PROPERTY FaultContactor : BOOL
GET
                    IF (Operational) THEN
	FaultContactor := lFaultContactor.Value;
ELSE
	FaultContactor := FALSE;	
END_IF
                  
END_GET
END_PROPERTY

PROPERTY FaultLevel : t_bms_fault_level
GET
                    IF (Operational) THEN
	FaultLevel := lFaultLevel.Value;
ELSE
	FaultLevel := cBMSFaultLevelNone;	
END_IF
                  
END_GET
END_PROPERTY

PROPERTY PackAverageTemperature : REAL
GET
                    PackAverageTemperature := lPackAverageTemperature.Value;

                  
END_GET
END_PROPERTY

PROPERTY PackChargeCurrent : REAL
GET
                    PackChargeCurrent := ABS(MIN(PackCurrent,0.0));


                  
END_GET
END_PROPERTY

PROPERTY PackChargeCurrentLimit : REAL
GET
                    IF (Operational) THEN // foobar should this be ValidTransmissions?
	PackChargeCurrentLimit := lPackChargeCurrentLimit.Value;
ELSE
	PackChargeCurrentLimit := 0.0;	
END_IF

                  
END_GET
END_PROPERTY

PROPERTY PackChargingCurrentTarget : REAL
GET
                    IF (Operational) THEN
	PackChargingCurrentTarget := lPackChargingCurrentTarget.Value;
ELSE
	PackChargingCurrentTarget := 0.0;	
END_IF


                  
END_GET
END_PROPERTY

PROPERTY PackChargingVoltageTarget : REAL
GET
                    PackChargingVoltageTarget := lPackChargingVoltageTarget.Value;

                  
END_GET
END_PROPERTY

PROPERTY PackCoolantTemperatureTarget : REAL
GET
                    PackCoolantTemperatureTarget := lPackCoolantTemperatureTarget.Value;
                  
END_GET
END_PROPERTY

PROPERTY PackCurrent : REAL
GET
                    IF (Operational) THEN
	PackCurrent := lPackCurrent.Value;
ELSE
	PackCurrent := 0.0;	
END_IF


                  
END_GET
END_PROPERTY

PROPERTY PackDischargeCurrent : REAL
GET
                    PackDischargeCurrent := MAX(PackCurrent,0.0);
                  
END_GET
END_PROPERTY

PROPERTY PackDischargeCurrentLimit : REAL
GET
                    IF (Operational) THEN
	PackDischargeCurrentLimit := lPackDischargeCurrentLimit.Value;
ELSE
	PackDischargeCurrentLimit := 0.0;	
END_IF


                  
END_GET
END_PROPERTY

PROPERTY PackFaultByte1 : USINT
GET
                    PackFaultByte1 := 0;
                  
END_GET
END_PROPERTY

PROPERTY PackFaultByte10 : USINT
GET
                    PackFaultByte10 := 0;
                  
END_GET
END_PROPERTY

PROPERTY PackFaultByte11 : USINT
GET
                    PackFaultByte11 := 0;
                  
END_GET
END_PROPERTY

PROPERTY PackFaultByte2 : USINT
GET
                    PackFaultByte2 := 0;
                  
END_GET
END_PROPERTY

PROPERTY PackFaultByte3 : USINT
GET
                    PackFaultByte3 := 0;
                  
END_GET
END_PROPERTY

PROPERTY PackFaultByte4 : USINT
GET
                    PackFaultByte4 := 0;
                  
END_GET
END_PROPERTY

PROPERTY PackFaultByte5 : USINT
GET
                    PackFaultByte5 := 0;
                  
END_GET
END_PROPERTY

PROPERTY PackFaultByte6 : USINT
GET
                    PackFaultByte6 := 0;
                  
END_GET
END_PROPERTY

PROPERTY PackFaultByte7 : USINT
GET
                    PackFaultByte7 := 0;
                  
END_GET
END_PROPERTY

PROPERTY PackFaultByte8 : USINT
GET
                    PackFaultByte8 := 0;
                  
END_GET
END_PROPERTY

PROPERTY PackFaultByte9 : USINT
GET
                    PackFaultByte9 := 0;
                  
END_GET
END_PROPERTY

PROPERTY PackFaultCode : USINT
GET
                    PackFaultCode := lPackFaultCode.Value;
                  
END_GET
END_PROPERTY

PROPERTY PackFaultNumber : USINT
GET
                    PackFaultNumber := lPackFaultNumber.Value;
                  
END_GET
END_PROPERTY

PROPERTY PackMaxTemperature : REAL
GET
                    PackMaxTemperature := lPackMaxTemperature.Value;
                  
END_GET
END_PROPERTY

PROPERTY PackMinTemperature : REAL
GET
                    PackMinTemperature := lPackMinTemperature.Value;
                  
END_GET
END_PROPERTY

PROPERTY PackSOC : t_percentage
GET
                    PackSOC := lPackSOC.Value;

                  
END_GET
END_PROPERTY

PROPERTY PackSOH : t_percentage
GET
                    PackSOH := lPackSOH.Value;
                  
END_GET
END_PROPERTY

PROPERTY PackTotalChargeEnergy : REAL
GET
                    PackTotalChargeEnergy := lPackTotalChargeEnergy.Value;
                  
END_GET
END_PROPERTY

PROPERTY PackTotalDischargeEnergy : REAL
GET
                    PackTotalDischargeEnergy := lPackTotalDischargeEnergy.Value;
                  
END_GET
END_PROPERTY

PROPERTY PackVoltage : REAL
GET
                    PackVoltage := lPackVoltage.Value;
                  
END_GET
END_PROPERTY

PROPERTY RequestDisconnect : BOOL
GET
                    RequestDisconnect := lRequestDisconnect.Value;
                  
END_GET
END_PROPERTY

PROPERTY RequestedBMSChargeState : t_bms_charge_state
GET
                    RequestedBMSChargeState := lRequestedBMSChargeState.Value;

                  
END_GET
SET
                    lRequestedBMSChargeState.Value := RequestedBMSChargeState;

                  
END_SET
END_PROPERTY

PROPERTY RequestedBMSState : t_bms_state
GET
                    RequestedBMSState := lRequestedBMSState.Value;
                  
END_GET
SET
                    lRequestedBMSState.Value := RequestedBMSState;


                  
END_SET
END_PROPERTY

PROPERTY RequestedTMSState : t_tms_state
GET
                    IF (Operational) THEN
	RequestedTMSState := lRequestedTMSState.Value;
ELSE
	RequestedTMSState := cTMSStateShutdown;	
END_IF
                  
END_GET
END_PROPERTY

PROPERTY TypeToken : t_medium_string
GET
                    TypeToken := 'cBMS';
                  
END_GET
END_PROPERTY

PROPERTY Peripheral : REFERENCE TO Peripheral
GET
                    Peripheral ref= lPeripheral;
                  
END_GET
END_PROPERTY
END_FUNCTION_BLOCK

FUNCTION_BLOCK ControllerCharger EXTENDS MimicCANOpenSlave
  VAR CONSTANT
    cChargingCurrentPhysicalMaxACSinglePhase : REAL := 38.0;  (* foobar changed from 48, CATL needs to allow higher values *)
    cOBCStatusPeriod : t_time := TIME#2s0ms;
  END_VAR
  VAR
    lChargingVoltageMax : ValueObjectRealOffsetScaledOutputReferenceUINTSwitched;
    lChargingCurrentMax : ValueObjectRealOffsetScaledOutputReferenceUINTSwitched;
    lHeatingMode : ValueObjectBoolOutputReferenceUSINT;
    lStopCharging : ValueObjectBoolOutputReferenceUSINT;
    lVoltage : ValueObjectRealScaledOffsetInputReferenceUINTSwitched;
    lCurrent : ValueObjectRealScaledOffsetInputReferenceUINTSwitched;
    lPower : ValueObjectRealScaledOffsetInputReferenceUSINT;
    lDiagnosticState : ValueObjectUINTInputReferenceUINT;
    lOBCStatus : ValueObjectEnumTypeInputReferenceUINT;
    lStatusCC : ValueObjectBoolInputReferenceUINT;
    lStatusCP : ValueObjectBoolInputReferenceUINT;
    lCurrentOBCState : ValueObjectEnumType;
    lRequestedOBCState : ValueObjectEnumType;
    lIgnoreOBCStatusNone : BOOL := TRUE;
    lChargingCurrentPhysicalMax : REAL := cChargingCurrentPhysicalMaxACSinglePhase;  (* foobar *)
    lOBCStatusTimer : t_timer;
    lOBCStatusDerived : t_obc_status;
  END_VAR

            ;
          

METHOD initialize
                  lChargingVoltageMax.Offset := 0.0;
lChargingVoltageMax.Scaling := 10.0;
lChargingVoltageMax.initializeValueObjectOp(OpSelf,'TargVoltage','Onboard charger target voltage','volts',cValueStyleConfigurable);

lChargingCurrentMax.Offset := 0.0;
lChargingCurrentMax.Scaling := 10.0;
lChargingCurrentMax.initializeValueObjectOp(OpSelf,'TargCurrent','Onboard charger target current','amps',cValueStyleConfigurable);

lHeatingMode.Index := 0;
lHeatingMode.initializeValueObjectOp(OpSelf,'Heating','Onboard charger heating mode','',cValueStyleConfigurable);

lStopCharging.Index := 0;
lStopCharging.initializeValueObjectOp(OpSelf,'Stop','Onboard charger stop status','',cValueStyleConfigurable);

lVoltage.Offset := 0.0;
lVoltage.Scaling := 0.1;
lVoltage.initializeValueObjectOp(OpSelf,'Voltage','Onboard charger measured voltage','volts',cValueStyleConfigurable);

lCurrent.Offset := 0.0;
lCurrent.Scaling := 0.1;
lCurrent.initializeValueObjectOp(OpSelf,'Current','Onboard charger measured current','amps',cValueStyleConfigurable);

lPower.Offset := 0.0;
lPower.Scaling := 100.0;
lPower.initializeValueObjectOp(OpSelf,'Power','Onboard charger measured power','kW',cValueStyleConfigurable);

lDiagnosticState.initializeValueObjectOp(OpSelf,'Diagnostic','Onboard charger current diagnostic','',cValueStyleConfigurable);

lStatusCC.Index := 5;
lStatusCC.initializeValueObjectOp(OpSelf,'CC','Onboard charger CC signal','',cValueStyleConfigurable);
lStatusCC.InputReference REF= lDiagnosticState.ValueReference;

lStatusCP.Index := 6;
lStatusCP.initializeValueObjectOp(OpSelf,'CP','Onboard charger CP signal','',cValueStyleConfigurable);
lStatusCP.InputReference REF= lDiagnosticState.ValueReference;

lOBCStatus.Index := 8;
lOBCStatus.Length := 2;
lOBCStatus.EnumType := cEnumTypeOBCStatus;
lOBCStatus.initializeValueObjectOp(OpSelf,'OBCStatus','Onboard charger OBC status','',cValueStyleConfigurable);
lOBCStatus.InputReference REF= lDiagnosticState.ValueReference;

lCurrentOBCState.EnumType := cEnumTypeOBCState;
lCurrentOBCState.initializeValueObject(NopSelf,'CrrOBCStt','Onboard charger current OBC state','',cValueStyleConfigurable);

lRequestedOBCState.EnumType := cEnumTypeOBCState;
lRequestedOBCState.initializeValueObject(NopSelf,'ReqOBCStt','Onboard charger requested OBC state','',cValueStyleConfigurable);
	
SUPER^.initialize();
SubSystem := cSubsystemBattery;

lAlarmCANOpenSlaveNotOperational.InitialSeverity := cSeverityNone;
lAlarmCANOpenSlaveNotOperational.SeverityWarningTimeout := T#250MS;
lAlarmCANOpenSlaveNotOperational.SeverityErrorTimeout := T#1S;
lAlarmCANOpenSlaveNotOperational.SeverityCriticalTimeout := T#5S;

lAlarmCANOpenSlaveAllowableUp.AllowableSystemState := cSystemStatePreparing;
lAlarmCANOpenSlaveAllowableUp.UpperSystemStateScope := cSystemStatePreparing;
lAlarmCANOpenSlaveAllowableUp.LowerSystemStateScope := cSystemStatePreparing;

lStartSystemStateScope := t_system_state.cSystemStatePreparing;
lOperationalSystemStateScopeLower := t_system_state.cSystemStateCharging;
lModulationSystemStateScope := t_system_state.cSystemStateCharging;

lModulationSeverity := cSeverityError; // foobar default or not?

lOBCStatusTimer.initialize();
lOBCStatusTimer.Enable := TRUE;
lOBCStatusTimer.Period := cOBCStatusPeriod;


                
END_METHOD

METHOD operator
                  SUPER^.operator();

setCurrentOBCState();

HeatingMode := FALSE;

CASE (RequestedOBCState) OF
	cOBCStateDisconnected:
		StopCharging := TRUE;	
	cOBCStateCharging:
		StopCharging := FALSE;
	cOBCStateStandby:
		StopCharging := TRUE;
	cOBCStateError:
		StopCharging := TRUE;
END_CASE

// lFaultHardware.Index := 0; 16#1
// lFaultTemperature.Index := 1; 16#2
// lFaultInputVoltage.Index := 2; 16#4
// lFaultBattery.Index := 3; 16#8
// lFaultCommunications.Index := 4; 16#10
// lWarningTemperature.Index := 14; 16#4000

// lStatusSwitch.Index := 12;
// lStatusFan.Index := 15;

IF (WORD_TO_BOOL(UINT_TO_WORD(lDiagnosticState.Value) AND 16#401F)) THEN
	lAlarmCANOpenSlaveNotify.triggerWithContext(UINT_TO_WORD(lDiagnosticState.Value));
END_IF


                
END_METHOD

METHOD setCurrentOBCState
                  IF (NOT(Operational)) THEN
	CurrentOBCState := cOBCStateDisconnected;
	RETURN;
END_IF

IF (OBCStatus<>cOBCStatusNone) THEN
	lOBCStatusTimer.reset();
END_IF
lOBCStatusTimer.operator();

IF (((NOT(lOBCStatusTimer.Expired)) OR
	(lIgnoreOBCStatusNone)) AND
	(OBCStatus=cOBCStatusNone)) THEN
	lOBCStatusDerived := cOBCStatusStandby ;
ELSE
	lOBCStatusDerived := OBCStatus;
END_IF

IF (lOBCStatusDerived=cOBCStatusNone) THEN
	CurrentOBCState := cOBCStateDisconnected;
	RETURN;
END_IF

IF (StatusCC) THEN
	CurrentOBCState := cOBCStateDisconnected;
	RETURN;
END_IF

CurrentOBCState := cOBCStateStandby;

IF ((NOT(StatusCC)) AND (StatusCP)) THEN
	// foobar not powered on
	RETURN;
END_IF

IF ((NOT(StatusCP)) AND
	(NOT(StatusCC)) AND
	(OBCStatus=cOBCStatusCharging) AND
	(lEnabled)) THEN
	CurrentOBCState := cOBCStateCharging;
END_IF

IF (OBCStatus=cOBCStatusError) THEN
	CurrentOBCState := cOBCStateError;
END_IF

                
END_METHOD

METHOD initializeCharger
  VAR_INPUT
    voltage : REFERENCE TO UINT;
    current : REFERENCE TO UINT;
    power : REFERENCE TO USINT;
    status : REFERENCE TO UINT;
    chargingVoltageMax : REFERENCE TO UINT;
    chargingCurrentMax : REFERENCE TO UINT;
    mode : REFERENCE TO USINT;
    command : REFERENCE TO USINT;
  END_VAR
                  lVoltage.InputReference REF= voltage;
lCurrent.InputReference REF= current;
lPower.InputReference REF= power;
lDiagnosticState.InputReference REF= status;

lChargingVoltageMax.OutputReference REF= chargingVoltageMax;
lChargingCurrentMax.OutputReference REF= chargingCurrentMax;
lHeatingMode.OutputReference REF= mode;
lStopCharging.OutputReference REF= command;

                
END_METHOD

PROPERTY ChargingCurrentMax : REAL
GET
                    ChargingCurrentMax := lChargingCurrentMax.Value;

                  
END_GET
SET
                    lChargingCurrentMax.Value := MIN(ChargingCurrentMax,lChargingCurrentPhysicalMax);
                  
END_SET
END_PROPERTY

PROPERTY ChargingVoltageMax : REAL
GET
                    ChargingVoltageMax := lChargingVoltageMax.Value;

                  
END_GET
SET
                    lChargingVoltageMax.Value := ChargingVoltageMax;
                  
END_SET
END_PROPERTY

PROPERTY Current : REAL
GET
                    Current := lCurrent.Value;

                  
END_GET
END_PROPERTY

PROPERTY CurrentOBCState : t_obc_state
GET
                    lCurrentOBCState.operator();
CurrentOBCState := lCurrentOBCState.Value;

                  
END_GET
SET
                    lCurrentOBCState.Value := CurrentOBCState;
                  
END_SET
END_PROPERTY

PROPERTY HeatingMode : BOOL
GET
                    HeatingMode := lHeatingMode.Value;

                  
END_GET
SET
                    lHeatingMode.Value := HeatingMode;
                  
END_SET
END_PROPERTY

(* {attribute 'monitoring' := 'call'} *)
PROPERTY OBCStatus : t_obc_status
GET
                    OBCStatus := lOBCStatus.Value;

                  
END_GET
END_PROPERTY

PROPERTY Power : REAL
GET
                    Power := lPower.Value;

                  
END_GET
END_PROPERTY

PROPERTY RequestedOBCState : t_obc_state
GET
                    lRequestedOBCState.operator();
RequestedOBCState := lRequestedOBCState.Value;
                  
END_GET
SET
                    lRequestedOBCState.Value := RequestedOBCState;


                  
END_SET
END_PROPERTY

(* {attribute 'monitoring' := 'call'} *)
PROPERTY StatusCC : BOOL
GET
                    StatusCC := lStatusCC.Value;

                  
END_GET
END_PROPERTY

(* {attribute 'monitoring' := 'call'} *)
PROPERTY StatusCP : BOOL
GET
                    StatusCP := lStatusCP.Value;

                  
END_GET
END_PROPERTY

PROPERTY StopCharging : BOOL
GET
                    StopCharging := lStopCharging.Value;

                  
END_GET
SET
                    lStopCharging.Value := StopCharging;

                  
END_SET
END_PROPERTY

PROPERTY TypeToken : t_medium_string
GET
                    TypeToken := 'cCharger';
                  
END_GET
END_PROPERTY

PROPERTY Voltage : REAL
GET
                    Voltage := lVoltage.Value;

                  
END_GET
END_PROPERTY
END_FUNCTION_BLOCK

FUNCTION_BLOCK ControllerChargerSlave EXTENDS ControllerCharger

            ;
          

METHOD initialize
                  SUPER^.initialize();

// invalid scope as only ChargerA controls AllowUp
lAlarmCANOpenSlaveAllowableUp.AllowableSystemState := cSystemStateCharging;
lAlarmCANOpenSlaveAllowableUp.UpperSystemStateScope := cSystemStateStandby;
lAlarmCANOpenSlaveAllowableUp.LowerSystemStateScope := cSystemStatePreparing;

lOperationalSystemStateScopeLower := t_system_state.cSystemStateCharging;
lOperationalSystemStateScopeUpper := t_system_state.cSystemStateCharging;

                
END_METHOD
END_FUNCTION_BLOCK

{attribute 'enable_dynamic_creation'}
FUNCTION_BLOCK ControllerMotor EXTENDS CANOpenSlave
  VAR_INPUT
    lRequestedThrottle : ValueObjectPercentage;
    lTypeSteer : BOOL := FALSE;
    lMaximumVelocity : REAL := 50.0;
    lAutomaticEnable : BOOL := TRUE;
    lAlwaysEnable : BOOL := FALSE;
  END_VAR
  VAR CONSTANT
    cStallPeriod : t_time := TIME#1s0ms;
    cNominalVoltage : REAL := 120.0;
    cTorquePeriod : t_time := TIME#250ms;
    cThrottleArbitrationAllowableDelta : t_percentage := 0.15;
    cThrottleArbitrationThreshold : t_percentage := 0.25;
    cThrottleArbitrationPeriod : t_time := TIME#2s0ms;
    cThrottleThreshold : t_percentage := 0.001;
    cThrottleFreeWheelThreshold : t_percentage := 0.002;
    cNMTDetectionPeriod : t_time := TIME#250ms;
    cEnabledPeriod : t_time := TIME#20s0ms;
    cMotorTemperatureType : DWORD := 4;
    cInitializeMotorHoldCount : USINT := 2;
    cInitializeMotorHoldPeriod : t_time := TIME#7s0ms;
    cNominalCurrent400A : REAL := 400.0;
    cPolePairs400A : REAL := 3.0;
    cControllerTemperatureInitialCutbackThreshold400A : REAL := 75.0;
    cControllerTemperatureCutoutThreshold400A : REAL := 100.0;
    cControllerTemperatureMinimumThreshold400A : t_percentage := 0.2;
    cMotorTemperatureInitialCutbackThreshold400A : REAL := 110.0;
    cMotorTemperatureCutoutThreshold400A : REAL := 160.0;
    cMotorTemperatureMinimumThreshold400A : t_percentage := 0.2;
    cMotorTemperatureInvalidRange400A : REAL := 200;
    cNominalCurrent150A : REAL := 150.0;
    cPolePairs150A : REAL := 2.0;
    cControllerTemperatureInitialCutbackThreshold150A : REAL := 75.0;
    cControllerTemperatureCutoutThreshold150A : REAL := 80.0;
    cControllerTemperatureMinimumThreshold150A : t_percentage := 0.2;
    cMotorTemperatureInitialCutbackThreshold150A : REAL := 110.0;
    cMotorTemperatureCutoutThreshold150A : REAL := 120.0;
    cMotorTemperatureMinimumThreshold150A : t_percentage := 0.2;
    cMotorTemperatureInvalidRange150A : REAL := 200;
  END_VAR
  VAR
    lVREnableStallAutomaticClearing : ValueReferenceBool;
    lEnableStallAutomaticClearing : BOOL := TRUE;
    lVREnableStallResponse : ValueReferenceBool;
    lEnableStallResponse : BOOL := FALSE;
    lVREnableHoldStationary : ValueReferenceBool;
    lEnableHoldStationary : BOOL := FALSE;
    lVREnableStallDetection : ValueReferenceBool;
    lEnableStallDetection : BOOL := FALSE;
    lVREnableThrottleArbitration : ValueReferenceBool;
    lEnableThrottleArbitration : BOOL := FALSE;
    lVREnableNMTDetectionTPDO : ValueReferenceBool;
    lEnableNMTDetectionTPDO : BOOL := FALSE;
    lVREnableInitializeHold : ValueReferenceBool;
    lEnableInitializeHold : BOOL := FALSE;
    lAlarmControllerTemperatureCutback : CutbackInterlock;
    lAlarmMotorTemperatureCutback : CutbackInterlock;
    lAlarmMotorTemperatureSensor : ReportableAlarm;
    lTargetSpeed : ValueObjectRealScaledOffsetOutputUINT;
    lEnable : ValueObjectBoolOutputUINT;
    lForward : ValueObjectBoolOutputUINT;
    lReverse : ValueObjectBoolOutputUINT;
    lClearAlarm : ValueObjectBoolOutputUINT;
    lVelocity : ValueObjectRealScaledOffsetInputReferenceINT;
    lTPDO1Stuffing : ValueObjectBoolInputReferenceUINT;
    lCurrent : ValueObjectRealScaledOffsetInputReferenceUSINT;
    lAlarm : ValueObjectUINTInputReferenceUINT;  (* foobar *)
    lMotorTemperature : ValueObjectRealScaledOffsetInputReferenceUSINT;
    lControllerTemperature : ValueObjectRealScaledOffsetInputReferenceSINT;
    lBatteryCurrent : ValueObjectRealScaledOffsetInputReferenceUSINT;
    lBatteryVoltage : ValueObjectRealScaledOffsetInputReferenceUINT;
    lBatteryPower : ValueObjectRealScaledOffset;
    lTorque : ValueObjectRealScaledOffsetInputUINT;  (* foobar *)
    lMotorTemperatureEnableCANSequence : MotorTemperatureEnableCANSequence;
    lCheckMotorTemperatureEnableCANMessage : CheckMotorTemperatureEnableCANMessage;
    lEnableRPDO1 : BOOL := TRUE;
    lTargetVelocity : REAL;
    lControl : WORD;
    lTorqueTimer : t_timer;
    lMotorTemperatureInvalidRange : REAL;
    lMotorTemperatureSensorRecovery : REAL;
    lEnableDiscriminatoryMotorTemperatureControl : BOOL := FALSE;  (* foobar *)
    lMotorTemperatureEnabled : BOOL := TRUE;
    lMotorTemperatureEnabledVerified : BOOL := FALSE;
    lHoldStationary : BOOL := FALSE;  (* lMaximumVelocity: REAL:= 50.0; lAutomaticEnable: BOOL:= TRUE; lAlwaysEnable: BOOL:= FALSE; *)
    lEnabledTimer : t_timer;
    lInitializeMotorHoldCounter : USINT := 0;
    lInitializeMotorHoldTimer : t_timer;
    lEnableFreeWheel : BOOL := FALSE;
    lFreeWheel : BOOL := FALSE;
    lDiagnostic : t_motor_diagnostic;
    _Diagnostic : t_motor_diagnostic;
    lStallTimer : t_timer;
    lStallState : t_stall_state := cStallStateNone;
    lStalled : BOOL := FALSE;
    lStallInput : BOOL := FALSE;
    lStalledCount : USINT := 0;
    lStationary : BOOL := FALSE;
    lTargetSpeedIndicator : USINT := 0;
    lZeroTargetSpeedIndicator : USINT := 0;
    lCurrentVelocityIndicator : USINT := 0;
    lZeroCurrentVelocityIndicator : USINT := 0;
    lStallIndicator : USINT := 0;
    lNoStallIndicator : USINT := 0;
    lStalledIndicator : USINT := 0;
    lNotStalledIndicator : USINT := 0;
    lRPDO1Message : T_x_can_msg;
    lSyncAlternateState : BOOL;
    lSDOTorque : CIA405.SDO_READ_DATA;
    lSDOTorqueData : DWORD;
    lSDOTorqueLastSuccessfulReadData : DWORD;
    lSDOTorqueDataLength : UDINT := 4;
    lSDOTorqueSuccess : BOOL := FALSE;
    lSDOTorqueAttemptCounter : USINT := 0;
    lSDOTorqueSuccessCounter : USINT := 0;
    lNominalVoltage : REAL := cNominalVoltage;
    lNominalCurrent : REAL := 0.0;
    lPolePairs : REAL := 1.0;
    lThrottleThreshold : t_percentage := cThrottleThreshold;
    lThrottleFreeWheelThreshold : t_percentage := cThrottleFreeWheelThreshold;
    lRequestedThrottlePrevious : t_percentage;
    lProposedThrottle : t_percentage;
    lMeasuredThrottle : t_percentage;
    lThrottleArbitrationDelta : t_percentage;
    lThrottleArbitrationAllowableDelta : t_percentage := cThrottleArbitrationAllowableDelta;
    lThrottleArbitrationThreshold : t_percentage := cThrottleArbitrationThreshold;
    lThrottleArbitrationTimer : t_timer;
    lRPDO1Alternate : BOOL := TRUE;
    lNMTDetectionTimer : t_timer;
    lTPDO1StuffingPrevious : BOOL;
  END_VAR

            ;
          

METHOD cancelSDOTorque
                  lSDOTorque.ENABLE := FALSE;
lSDOTorqueDataLength := 4;
lSDOTorque(DATALENGTH:=lSDOTorqueDataLength);

                
END_METHOD

METHOD checkMotorTemperatureEnabled
                  //requestSDORead(TRUE,16#20F1,2,4);

IF (lCheckMotorTemperatureEnableCANMessage.Success) THEN
	lMotorTemperatureEnabledVerified := TRUE;
	lMotorTemperatureEnabled := lCheckMotorTemperatureEnableCANMessage.MotorTemperatureEnabled;
	lCheckMotorTemperatureEnableCANMessage.reset();
	RETURN;
END_IF

IF (NOT(lCheckMotorTemperatureEnableCANMessage.Running)) THEN
	lCheckMotorTemperatureEnableCANMessage.start();
END_IF


                
END_METHOD

METHOD emergencyHandler
  VAR_INPUT
    info : t_canopen_emcy;
  END_VAR
  VAR
    eid : t_motor_emcy_id;
    first : BOOL;
  END_VAR
                  first := emergencyRegisterAdd(info);

eid := WORD_TO_INT(info.EMCY_ERROR_CODE);

CASE eid OF
	t_motor_emcy_id.cEMCY_none:
		RETURN;

	t_motor_emcy_id.cEMCY_CONTACTOR_OPEN,
	t_motor_emcy_id.cEMCY_CONTACTOR_CLOSED,
	t_motor_emcy_id.cEMCY_PUMP_VMN_LOW,
	t_motor_emcy_id.cEMCY_PUMP_VMN_HIGH,
	t_motor_emcy_id.cEMCY_TILLER_ERROR,
	t_motor_emcy_id.cEMCY_PUMP_VMN_NOT_OK,
	t_motor_emcy_id.cEMCY_HVIL_FAIL,
	t_motor_emcy_id.cEMCY_SEAT_MISMATCH,
	t_motor_emcy_id.cEMCY_PEDAL_WIRE_KO,
	t_motor_emcy_id.cEMCY_PUMP_VACC_NOT_OK,
	t_motor_emcy_id.cEMCY_PUMP_INC_START,
	t_motor_emcy_id.cEMCY_PUMP_VACC_RANGE,
	t_motor_emcy_id.cEMCY_HANDBRAKE:
		lAlarmCANOpenSlaveNotify.triggerWithContext(INT_TO_LWORD(eid));
		RETURN;
				
	t_motor_emcy_id.cEMCY_MC_EB_COIL_SHORT,
	t_motor_emcy_id.cEMCY_DRIVER_SHORTED,
	t_motor_emcy_id.cEMCY_CONTACTOR_DRIVER,
	t_motor_emcy_id.cEMCY_EVP_DRIV_SHORT,
	t_motor_emcy_id.cEMCY_EVP_COIL_SHORT,
	t_motor_emcy_id.cEMCY_EVP2_COIL_SHORT,
	t_motor_emcy_id.cEMCY_HW_FAULT_MC,
	t_motor_emcy_id.cEMCY_POSITIVE_LC_OPEN,
	t_motor_emcy_id.cEMCY_LC_COIL_OPEN,
	t_motor_emcy_id.cEMCY_CONTROLLER_MISM,
	t_motor_emcy_id.cEMCY_NO_CAN_MSG,
	t_motor_emcy_id.cEMCY_WRONG_SET_BAT,
	t_motor_emcy_id.cEMCY_WRONG_KEY_VOLT,
	t_motor_emcy_id.cEMCY_CAPACITOR_CHARGE,
	t_motor_emcy_id.cEMCY_WRONG_FBSENSSET,
	t_motor_emcy_id.cEMCY_OFFSET_SPDSENS,
	t_motor_emcy_id.cEMCY_SPEED_OVERHEAD,
	t_motor_emcy_id.cEMCY_WRONG_RAM_MEM,
	t_motor_emcy_id.cEMCY_POWER_MISMATCH,
	t_motor_emcy_id.cEMCY_IQ_MISMATCHED,
	t_motor_emcy_id.cEMCY_FIELD_ORIENT_KO,
	t_motor_emcy_id.cEMCY_WATCHDOG,
	t_motor_emcy_id.cEMCY_SAFETY_INIT_XX,
	t_motor_emcy_id.cEMCY_SAFETY_SW_XX,
	t_motor_emcy_id.cEMCY_SAFETY_DIAG_XX,
	t_motor_emcy_id.cEMCY_STBY_HIGH,
	t_motor_emcy_id.cEMCY_VMN_HIGH,
	t_motor_emcy_id.cEMCY_INIT_VMN_HIGH,
	t_motor_emcy_id.cEMCY_VMN_LOW,
	t_motor_emcy_id.cEMCY_INIT_VMN_LOW,
	t_motor_emcy_id.cEMCY_POS_EB_SHORTED,
	t_motor_emcy_id.cEMCY_SMARTDRIVER_KO,
	t_motor_emcy_id.cEMCY_AUX_BATT_SHORT,
	t_motor_emcy_id.cEMCY_VKEY_OFF_SHORTED,
	t_motor_emcy_id.cEMCY_LOGIC_FAILURE_1,
	t_motor_emcy_id.cEMCY_LOGIC_FAILURE_3,
	t_motor_emcy_id.cEMCY_LOGIC_FAILURE_2,
	t_motor_emcy_id.cEMCY_SENSOR_SUPPLY_XX,
	t_motor_emcy_id.cEMCY_POSEBSHORT_PIN,
	t_motor_emcy_id.cEMCY_ED_SLIP_MISMATCH,
	t_motor_emcy_id.cEMCY_POSEBSHORT_GND,
	t_motor_emcy_id.cEMCY_SHORT_CIRCUIT_KO,
	t_motor_emcy_id.cEMCY_SHORT_CIRCUIT,
	t_motor_emcy_id.cEMCY_IMS_ERROR,
	t_motor_emcy_id.cEMCY_SPEED_FBERR_XX,
	t_motor_emcy_id.cEMCY_MOTPHASE_SH,
	t_motor_emcy_id.cEMCY_VDC_OFF_SHORTED,
	t_motor_emcy_id.cEMCY_HW_FAULT,
	t_motor_emcy_id.cEMCY_POWERMOS_SHORTED,
	t_motor_emcy_id.cEMCY_CTRAP_THRESHOLD,
	t_motor_emcy_id.cEMCY_OUT_MISMATCH_PU,
	t_motor_emcy_id.cEMCY_SP_MISMATCH_XX,
	t_motor_emcy_id.cEMCY_ANALOG_INPUT,
	t_motor_emcy_id.cEMCY_OVERLOAD,
	t_motor_emcy_id.cEMCY_VDC_LINK_OVERV:
		lAlarmCANOpenSlaveBlock.triggerWithContext(INT_TO_LWORD(eid));
		RETURN;
		
	t_motor_emcy_id.cEMCY_EB_DRIVSHRT,
	t_motor_emcy_id.cEMCY_EB_DRIVOPEN,
	t_motor_emcy_id.cEMCY_EVP_COIL_OPEN,
	t_motor_emcy_id.cEMCY_VACC_NOT_OK,
	t_motor_emcy_id.cEMCY_BMS_NOT_READY,
	t_motor_emcy_id.cEMCY_POT_MISMATCH,
	t_motor_emcy_id.cEMCY_AGV,
	t_motor_emcy_id.cEMCY_REMA_T_ALARM,
	t_motor_emcy_id.cEMCY_SENS_BAT_TEMP_KO,
	t_motor_emcy_id.cEMCY_EMERGENCY,
	t_motor_emcy_id.cEMCY_LIFT_LOWER,
	t_motor_emcy_id.cEMCY_PARAM_TRANSFER,
	t_motor_emcy_id.cEMCY_EPS_RELAY_OPEN,
	t_motor_emcy_id.cEMCY_EB_COIL_OPEN,
	t_motor_emcy_id.cEMCY_PEB_PEVP_NOT_OK,
	t_motor_emcy_id.cEMCY_PEV_NOT_OK,
	t_motor_emcy_id.cEMCY_VACC_OUT_RANGE,
	t_motor_emcy_id.cEMCY_HW_FAULT_EB,
	t_motor_emcy_id.cEMCY_CONT_DRV_EV,
	t_motor_emcy_id.cEMCY_COIL_SHOR_EVAUX,
	t_motor_emcy_id.cEMCY_EVP_DRIVER_OPEN,
	t_motor_emcy_id.cEMCY_DRV_SHOR_EV,
	t_motor_emcy_id.cEMCY_NO_CAN_WR_MSGXX,
	t_motor_emcy_id.cEMCY_STO_SS1_ALARM_XX,
	t_motor_emcy_id.cEMCY_WRONG_PERFORM,
	t_motor_emcy_id.cEMCY_WRONG_SLAVE_VER,
	t_motor_emcy_id.cEMCY_MS_PAR_CHK_MISM,
	t_motor_emcy_id.cEMCY_CURRENT_PROFILE,
	t_motor_emcy_id.cEMCY_EEPROM_KO,
	t_motor_emcy_id.cEMCY_COIL_SHOR_EB,
	t_motor_emcy_id.cEMCY_STO_SS1_ACTIVEXX,
	t_motor_emcy_id.cEMCY_RPM_HIGH,
	t_motor_emcy_id.cEMCY_STALL_ROTOR,
	t_motor_emcy_id.cEMCY_INCORRECT_START,
	t_motor_emcy_id.cEMCY_FORW_BACK,
	t_motor_emcy_id.cEMCY_MOTOR_TEMP_STOP:
		lAlarmCANOpenSlaveBlock.triggerWithContext(INT_TO_LWORD(eid));
		IF (first) THEN
			lAlarmCANOpenSlaveStop.triggerWithContext(INT_TO_LWORD(eid));
		END_IF
	
		RETURN;
		
	t_motor_emcy_id.cEMCY_THERMIC_SENS_KO,
	t_motor_emcy_id.cEMCY_THERMPUSENSKO,
	t_motor_emcy_id.cEMCY_SENS_MOT_TEMP_KO:
		lAlarmCANOpenSlaveBlock.triggerWithContext(INT_TO_LWORD(eid));; //foobar disable remedy
		RETURN;
END_CASE

lAlarmCANOpenSlaveNotify.triggerWithContext(INT_TO_LWORD(eid));

	//t_motor_emcy_id.cEMCY_REMA_T_ALARM,								//duplicate id
	//	lAlarmCANOpenStop.triggerWithContext(eid);

	//t_motor_emcy_id.cEMCY_SP_MISMATCH_PUMP,                     //duplicate id
	//	lAlarmCANOpenSlaveBlock.triggerWithContext(eid);
	
	//t_motor_emcy_id.cEMCY_OPEN_COIL_EV,							//duplicate id
	//	lAlarmCANOpenStop.triggerWithContext(eid);
	
	//t_motor_emcy_id.cEMCY_WRONG_FBSENSSET,					//duplicate id
	//	lAlarmCANOpenSlaveBlock.triggerWithContext(eid);
		
	//t_motor_emcy_id.cEMCY_WSET_TG_EB_XX,						//duplicate id
	//	lAlarmCANOpenSlaveBlock.triggerWithContext(eid);
	
	//t_motor_emcy_id.cEMCY_INPUT_MISMATCH,						//duplicate id
	//	lAlarmCANOpenSlaveBlock.triggerWithContext(eid);
		
	//t_motor_emcy_id.cEMCY_SAFETY_DIAG_XX,						//duplicate
	//	lAlarmCANOpenSlaveBlock.triggerWithContext(eid);
	
	//t_motor_emcy_id.cEMCY_SAFETY_SW_XX,							//duplicate
	//	lAlarmCANOpenSlaveBlock.triggerWithContext(eid);
	
	//t_motor_emcy_id.cEMCY_SAFETY_INIT_XX,						//duplicate
	//	lAlarmCANOpenSlaveBlock.triggerWithContext(eid);
	
	//t_motor_emcy_id.cEMCY_OUT_MISMATCH_XX,				duplicate label
	//	lAlarmCANOpenSlaveBlock.triggerWithContext(eid);
	
	//t_motor_emcy_id.cEMCY_STO_SS1_ALARM_XX,					duplicate label
	//	lEventHandlerOperatingBlockingFault.operator(eid,controller,info);
	

                
END_METHOD

METHOD initialize
                  IF (lTypeSteer) THEN
	lNominalCurrent := cNominalCurrent150A;
	lPolePairs := cPolePairs150A;

	lMotorTemperatureInvalidRange := cMotorTemperatureInvalidRange150A;
	lMotorTemperatureSensorRecovery := cMotorTemperatureInvalidRange150A;
ELSE
	lNominalCurrent := cNominalCurrent400A;
	lPolePairs := cPolePairs400A;

	lMotorTemperatureInvalidRange := cMotorTemperatureInvalidRange400A;
	lMotorTemperatureSensorRecovery := cMotorTemperatureInvalidRange400A;
END_IF

lVREnableStallAutomaticClearing.initializeValueReference(lEnableStallAutomaticClearing,NopSelf,'EnblStallClr','Stall states are automatically cleared','',cValueStyleParameter);
lVREnableStallResponse.initializeValueReference(lEnableStallResponse,NopSelf,'EnbleStallResp','Automatically handle stall states','',cValueStyleParameter);
lVREnableHoldStationary.initializeValueReference(lEnableHoldStationary,NopSelf,'EnbleHoldStat','Hold on stationary','',cValueStyleParameter);
lVREnableStallDetection.initializeValueReference(lEnableStallDetection,NopSelf,'EnbleStallDet','Stall states are automatically detected','',cValueStyleParameter);
lVREnableThrottleArbitration.initializeValueReference(lEnableThrottleArbitration,NopSelf,'EnblThrttArb','Enable throttle arbitration','',cValueStyleParameter);
lVREnableNMTDetectionTPDO.initializeValueReference(lEnableNMTDetectionTPDO,NopSelf,'EnbleNMTDet','Detect NMT state from TPOD traffic','',cValueStyleParameter);
lVREnableInitializeHold.initializeValueReference(lEnableInitializeHold,NopSelf,'EnblInitHold','Enable initial hold strategy','',cValueStyleParameter);

lAlarmControllerTemperatureCutback.initializeState(NopSelf,'',cACControllerTemperatureCutback);
lAlarmControllerTemperatureCutback.Qualifier := cChargeQualifierBoth;

lAlarmMotorTemperatureCutback.initializeState(NopSelf,'',cACMotorTemperatureCutback);
lAlarmMotorTemperatureCutback.Qualifier := cChargeQualifierBoth;

lAlarmMotorTemperatureSensor.initializeState(NopSelf,'',cACMotorTemperatureSensor);
lAlarmMotorTemperatureSensor.Life := 10;

lTargetSpeed.Scaling := 10.0 * lPolePairs;
lTargetSpeed.initializeValueObject(NopSelf,'TargetSpeed','Motor target speed','rpm',cValueStyleConfigurable);

lEnable.Index := 0;
lEnable.initializeValueObject(NopSelf,'EnableMotor','Motor enable state','',cValueStyleConfigurable);

lForward.Index := 3;
lForward.initializeValueObject(NopSelf,'Forward','Motor forward state','',cValueStyleConfigurable);

lReverse.Index := 4;
lReverse.initializeValueObject(NopSelf,'Reverse','Motor reverse state','',cValueStyleConfigurable);

lClearAlarm.Index := 13;
lClearAlarm.initializeValueObject(NopSelf,'ClearAlarm','Motor clear alarm state','',cValueStyleConfigurable);

lVelocity.Scaling := 0.1 / lPolePairs;
lVelocity.initializeValueObjectOp(OpSelf,'Velocity','Motor current velocity','rpm',cValueStyleConfigurable);

lTPDO1Stuffing.Index := 15;
lTPDO1Stuffing.initializeValueObjectOp(OpSelf,'TPO1Stuffing','Motor TPOD stuffing state','',cValueStyleConfigurable);

lCurrent.Scaling := lNominalCurrent/200.0;
lCurrent.initializeValueObjectOp(OpSelf,'Current','Motor measured current','amps',cValueStyleConfigurable);

lAlarm.initializeValueObjectOp(OpSelf,'Alarm','Motor alarm state','',cValueStyleConfigurable);

lMotorTemperature.Offset := -40;
lMotorTemperature.initializeValueObjectOp(OpSelf,'MotorTemp','Motor temperature','celcius',cValueStyleConfigurable);

lControllerTemperature.initializeValueObjectOp(OpSelf,'CntrlTemp','Controller temperature','celcius',cValueStyleConfigurable);

lBatteryCurrent.Scaling := lNominalCurrent/127.0;//foobar usint not sint, requires offset?
lBatteryCurrent.initializeValueObjectOp(OpSelf,'BattCurrent','Motor battery current','amps',cValueStyleConfigurable);

lBatteryVoltage.Scaling := 0.001*lNominalVoltage;
lBatteryVoltage.initializeValueObjectOp(OpSelf,'BattVoltage','Motor battery voltage','volts',cValueStyleConfigurable);

lBatteryPower.Scaling := 0.001;
lBatteryPower.Offset := 0.0;
lBatteryPower.initializeValueObjectOp(OpSelf,'BattPower','Motor battery power','kW',cValueStyleConfigurable);

lTorque.initializeValueObject(NopSelf,'Torque','Motor current torque','Nm',cValueStyleConfigurable);

SUPER^.initialize();

lStallTimer.Enable := TRUE;
lStallTimer.Period := cStallPeriod;
lStallTimer.initialize();

lTorqueTimer.initialize();
lTorqueTimer.Enable := TRUE;
lTorqueTimer.Period := cTorquePeriod;

lThrottleArbitrationTimer.initialize();
lThrottleArbitrationTimer.Enable := TRUE;
lThrottleArbitrationTimer.Period := cThrottleArbitrationPeriod;

lRPDO1Message.t_Id.u32_Id := 16#200 + lControllerId;
lRPDO1Message.t_Id.u8_Xtd := X_OFF;
lRPDO1Message.u8_Dlc := 8;
lRPDO1Message.au8_Data[0] := 0;
lRPDO1Message.au8_Data[1] := 0;
lRPDO1Message.au8_Data[2] := 0;
lRPDO1Message.au8_Data[3] := 0;
lRPDO1Message.au8_Data[4] := 0;
lRPDO1Message.au8_Data[5] := 0;
lRPDO1Message.au8_Data[6] := 0;
lRPDO1Message.au8_Data[7] := 0;

lSDORead.DEVICE := lControllerId + 2;
lSDOWrite.DEVICE := lControllerId + 2;

lSDOTorque.DEVICE := lControllerId + 2;
lSDOTorque.CHANNEL := 0;
lSDOTorque.NETWORK := lNetworkId;
lSDOTorque.ENABLE := FALSE;
lSDOTorque.TIMEOUT := 500;
lSDOTorque.MODE := CIA405.SDO_MODE.AUTO;
lSDOTorque.DATA := ADR(lSDOTorqueData);

lNMTDetectionTimer.initialize();
lNMTDetectionTimer.Enable := TRUE;
lNMTDetectionTimer.Period := cNMTDetectionPeriod;

lEnabledTimer.initialize();
lEnabledTimer.Enable := TRUE;
lEnabledTimer.Period := cEnabledPeriod;

lMotorTemperatureEnableCANSequence.initialize();
lCheckMotorTemperatureEnableCANMessage.initialize();

lInitializeMotorHoldTimer.initialize();
lInitializeMotorHoldTimer.Enable := TRUE;
lInitializeMotorHoldTimer.Period := cInitializeMotorHoldPeriod;

IF (lTypeSteer) THEN
	lAlarmControllerTemperatureCutback.InitialCutbackThreshold := cControllerTemperatureInitialCutbackThreshold150A;
	lAlarmControllerTemperatureCutback.CutoutThreshold := cControllerTemperatureCutoutThreshold150A;
	lAlarmControllerTemperatureCutback.MinimiumThreshold := cControllerTemperatureMinimumThreshold150A;

	lAlarmMotorTemperatureCutback.InitialCutbackThreshold := cMotorTemperatureInitialCutbackThreshold150A;
	lAlarmMotorTemperatureCutback.CutoutThreshold := cMotorTemperatureCutoutThreshold150A;
	lAlarmMotorTemperatureCutback.MinimiumThreshold := cMotorTemperatureMinimumThreshold150A;
	
	lAlarmCANOpenSlaveModulation.registerServer(gSystemPrimary.Travel.Interlock);
	lAlarmCANOpenSlaveBlock.registerServer(gSystemPrimary.Travel.Interlock);

	lAlarmControllerTemperatureCutback.registerServer(gSystemPrimary.Travel.ChargeInterlock);
	lAlarmMotorTemperatureCutback.registerServer(gSystemPrimary.Travel.ChargeInterlock);

	lMaximumVelocity := cSteerMotorMaximumVelocityAsHz;

	lAlwaysEnable := FALSE;
	lAutomaticEnable := TRUE;
ELSE
	lAlarmControllerTemperatureCutback.InitialCutbackThreshold := cControllerTemperatureInitialCutbackThreshold400A;
	lAlarmControllerTemperatureCutback.CutoutThreshold := cControllerTemperatureCutoutThreshold400A;
	lAlarmControllerTemperatureCutback.MinimiumThreshold := cControllerTemperatureMinimumThreshold400A;

	lAlarmMotorTemperatureCutback.InitialCutbackThreshold := cMotorTemperatureInitialCutbackThreshold400A;
	lAlarmMotorTemperatureCutback.CutoutThreshold := cMotorTemperatureCutoutThreshold400A;
	lAlarmMotorTemperatureCutback.MinimiumThreshold := cMotorTemperatureMinimumThreshold400A;
END_IF

                
END_METHOD

METHOD initializeMotorHold
                  lInitializeMotorHoldCounter := cInitializeMotorHoldCount;

lInitializeMotorHoldTimer.reset();

                
END_METHOD

METHOD operator
                  SUPER^.operator();

IF (gSystemPrimary.SystemState.State<>cSystemStateOperational) THEN
	RequestedThrottle := 0.0;
	Diagnostic := cMotorDiagnosticNotOperational;
END_IF

IF (NOT(gSystemPrimary.OperatingMode.Ready)) THEN
	RequestedThrottle := 0.0;
	Diagnostic := cMotorDiagnosticOperatingMode;
END_IF

IF (HoldStationary) THEN
	RequestedThrottle := 0.0;
	Diagnostic := cMotorDiagnosticHoldStationary;	
END_IF

IF (NOT(Enabled)) THEN
	RequestedThrottle := 0.0;
	Diagnostic := cMotorDiagnosticDisabled;
END_IF

lRequestedThrottlePrevious := RequestedThrottle;
lProposedThrottle := lRequestedThrottlePrevious;
lMeasuredThrottle := velocityToThrottle(Velocity);

stallManagement();
throttleArbitration();

lFreeWheel := ((lEnableFreeWheel) AND (ABS(lProposedThrottle)<lThrottleFreeWheelThreshold));
lEnableFreeWheel := FALSE;

IF (ABS(lProposedThrottle)<lThrottleThreshold) THEN
	lProposedThrottle := 0.0;
END_IF

IF (lAlwaysEnable) THEN
	lEnable.Value := NOT(lFreeWheel);

ELSIF (lAutomaticEnable) THEN
	IF (lProposedThrottle<>0) THEN
		lEnabledTimer.reset();
	END_IF	
	IF ((lHoldStationary) AND (lEnableHoldStationary)) THEN
		lEnabledTimer.reset();
	END_IF
	lEnabledTimer.operator();

	lEnable.Value := ((Enabled) AND
		(gSystemPrimary.SystemState.State>=cSystemStateExitOperational) AND
		(NOT(lEnabledTimer.Expired)) AND
		(NOT(lFreeWheel)));

ELSE
	lEnable.Value := Enabled;	

END_IF

lTargetVelocity := throttleToVelocity(lProposedThrottle);

IF (lEnableInitializeHold) THEN
	lInitializeMotorHoldTimer.operator();
	
	IF (lTargetVelocity=0) THEN
		IF (lInitializeMotorHoldTimer.Expired) THEN
			initializeMotorHold();
		END_IF
	ELSE
		lInitializeMotorHoldTimer.reset();
	END_IF

	IF (lInitializeMotorHoldCounter>0) THEN
		lInitializeMotorHoldCounter := lInitializeMotorHoldCounter - 1;
			
		IF (lTargetVelocity=0) THEN
			lTargetVelocity := 0.1/lPolePairs;
			Diagnostic := cMotorDiagnosticInitializeHold;
		END_IF
	END_IF
END_IF

IF (NOT(lEnable.Value)) THEN
	lForward.Value := FALSE;
	lReverse.Value := FALSE;
ELSE
	IF (lTargetVelocity = 0) THEN
		// forward and reverse carry forward from previous
		// ensure both are not active at the same time, at least one is active

		IF (lForward.Value) THEN
			lReverse.Value := FALSE;
		END_IF
		IF (lReverse.Value) THEN
			lForward.Value := FALSE;
		END_IF
		IF ((NOT(lForward.Value)) AND (NOT(lReverse.Value))) THEN
			lForward.Value := TRUE;		
		END_IF
	ELSE
		lForward.Value := (lTargetVelocity > 0);
		lReverse.Value := (lTargetVelocity < 0);
	END_IF
END_IF

lTargetSpeed.Value := ABS(lTargetVelocity);
lStationary := ((Velocity=0) AND (TargetSpeed=0));

rpdo1();

IF ((lTorqueTimer.Enable) AND 
	(RequestedThrottle<>0.0)) THEN
	lTorqueTimer.operator();
	IF (lTorqueTimer.Expired) THEN
		lTorqueTimer.reset();
		requestSDOTorque();
	END_IF
	IF (lSDOTorqueSuccess) THEN
		lTorque.Input := DWORD_TO_UINT(lSDOLastSuccessfulReadData);
		lSDOTorqueSuccess := FALSE;
	END_IF
ELSE
	lTorque.Input := 0; //foobar check sdo are we getting real values
END_IF

IF (lSDOTorque.ENABLE) THEN
	lSDOTorque(DATALENGTH:=lSDOTorqueDataLength);
	IF ((lSDOTorque.CONFIRM) OR (lSDORead.ERROR<>CIA405.CANOPEN_KERNEL_ERROR.CANOPEN_KERNEL_NO_ERROR)) THEN
		lSDOTorque.ENABLE := FALSE;
		lSDOTorqueAttemptCounter := lSDOTorqueAttemptCounter + 1;
		IF (lSDOTorque.CONFIRM) THEN
			lSDOTorqueSuccess := TRUE;
			lSDOTorqueLastSuccessfulReadData := lSDOTorqueData;
			lSDOTorqueSuccessCounter := lSDOTorqueSuccessCounter + 1;
		END_IF
	END_IF	
END_IF

lMotorTemperatureEnableCANSequence.operator(); // foobar deprecated?
lCheckMotorTemperatureEnableCANMessage.operator(); // foobar deprecated?

lAlarmControllerTemperatureCutback.Value := ControllerTemperature;
lAlarmControllerTemperatureCutback.test(FALSE);

IF (MotorTemperature>=lMotorTemperatureInvalidRange) THEN
	lAlarmMotorTemperatureSensor.trigger(FALSE);
	lAlarmMotorTemperatureCutback.Value := lMotorTemperatureSensorRecovery;
ELSE
	lAlarmMotorTemperatureCutback.Value := MotorTemperature;
END_IF
lAlarmMotorTemperatureCutback.test(FALSE);

lBatteryPower.Value := lBatteryCurrent.Value * lBatteryVoltage.Value;

lDiagnostic := _Diagnostic;
_Diagnostic := cMotorDiagnosticOK;

                
END_METHOD

METHOD requestSDOTorque
                  cancelSDOTorque();

lSDOTorque.ENABLE := TRUE;

lSDOTorque.INDEX := 16#210E;
lSDOTorque.SUBINDEX := 0;
lSDOTorqueDataLength := 2;

lSDOTorqueSuccess := FALSE;

                
END_METHOD

METHOD rpdo1
                  IF (NOT(lEnableRPDO1)) THEN
	RETURN;
END_IF

lControl := ((2) OR
	(UINT_TO_WORD(lEnable.Output)) OR
	(UINT_TO_WORD(lForward.Output)) OR
	(UINT_TO_WORD(lReverse.Output)) OR
	(UINT_TO_WORD(lClearAlarm.Output)) OR //foobar clearing and recovering from alarms
	SHL(BOOL_TO_WORD(lSyncAlternateState),15));

lRPDO1Message.au8_Data[0] := UINT_TO_BYTE(lTargetSpeed.Output);
lRPDO1Message.au8_Data[1] := WORD_TO_BYTE(SHR(UINT_TO_WORD(lTargetSpeed.Output),8));
lRPDO1Message.au8_Data[2] := UINT_TO_BYTE(lControl);
lRPDO1Message.au8_Data[3] := WORD_TO_BYTE(SHR(UINT_TO_WORD(lControl),8));

IF (lMaster.TransmitMessage.transmit(lRPDO1Message)=C_OVERFLOW) THEN
	lOverflowCounter := lOverflowCounter + 1;
ELSE
	lSyncAlternateState := NOT(lSyncAlternateState);
END_IF

                
END_METHOD

METHOD sdoReadHandler
                  IF (lSDORead.INDEX=16#20F1) THEN
	lMotorTemperatureEnabled := (lSDOReadData<>0);
	lMotorTemperatureEnabledVerified := TRUE;
END_IF
                
END_METHOD

METHOD stallDetection
                  IF (NOT(lEnableStallDetection)) THEN
	lStalled := lStallInput := FALSE;
	RETURN;
END_IF

lStallInput := ((Velocity=0) AND (TargetSpeed>0)); // foobar no reportable for stall detection

IF (TargetSpeed=0) THEN
	lZeroTargetSpeedIndicator := lZeroTargetSpeedIndicator + 1;
	lTargetSpeedIndicator := 0;
ELSE
	lTargetSpeedIndicator := lTargetSpeedIndicator + 1;
	lZeroTargetSpeedIndicator := 0;	
END_IF

IF (Velocity=0) THEN
	lZeroCurrentVelocityIndicator := lZeroCurrentVelocityIndicator + 1;
	lCurrentVelocityIndicator := 0;
ELSE
	lCurrentVelocityIndicator := lCurrentVelocityIndicator + 1;
	lZeroCurrentVelocityIndicator := 0;	
END_IF

IF (NOT(lStallInput)) THEN
	lStallTimer.reset();
	lNoStallIndicator := lNoStallIndicator + 1;
	lStallIndicator := 0;
ELSE
	lStallIndicator := lStallIndicator + 1;
	lNoStallIndicator := 0;
END_IF

lStallTimer.operator();
IF ((lStallInput) AND (lStallTimer.Expired)) THEN
	IF (NOT(lStalled)) THEN
		lStalledCount := lStalledCount + 1;
	END_IF

	lStalled := TRUE;
ELSE
	lStalled := FALSE;
END_IF

IF (lStalled) THEN
	lStalledIndicator := lStalledIndicator + 1;
	lNotStalledIndicator := 0;
ELSE
	lNotStalledIndicator := lNotStalledIndicator + 1;
	lStalledIndicator := 0;
END_IF

                
END_METHOD

METHOD stallManagement
                  stallDetection();

CASE lStallState OF
	cStallStateNone:
		IF (Stalled) THEN
			lStallState := cStallStateDetected;
		END_IF

	cStallStateDetected:		
		lStallState := cStallStateCurrent;

	cStallStateCurrent:
		IF (NOT(Stalled)) THEN
			IF (lEnableStallAutomaticClearing) THEN
				lStallState := cStallStateNone;
			ELSE
				lStallState := cStallStateClearing;
			END_IF
		END_IF
		
	cStallStateClearing:
		lStallState := cStallStateNone;
END_CASE

IF ((lStallState>cStallStateNone) AND
	(lEnableStallResponse)) THEN
	stallResponse();
END_IF

                
END_METHOD

METHOD stallResponse
                  lProposedThrottle := 0.0;
Diagnostic := cMotorDiagnosticStalled;
                
END_METHOD

METHOD startHandler
                  SUPER^.startHandler();

IF ((lEnableDiscriminatoryMotorTemperatureControl) AND
	(NOT(lMotorTemperatureEnabledVerified))) THEN
	checkMotorTemperatureEnabled();
END_IF
                
END_METHOD

METHOD startResetHandler
                  lMotorTemperatureEnabledVerified := FALSE;
lCheckMotorTemperatureEnableCANMessage.reset();
                
END_METHOD

METHOD throttleArbitration
                  IF (lEnableThrottleArbitration) THEN
	IF (lRequestedThrottlePrevious<>RequestedThrottle) THEN
		lThrottleArbitrationTimer.reset();
	END_IF

	lThrottleArbitrationTimer.operator();
	
	IF ((ABS(RequestedThrottle)>lThrottleArbitrationThreshold) AND
		(lThrottleArbitrationTimer.Expired) AND
		(((RequestedThrottle>0) AND (lMeasuredThrottle>0)) OR ((RequestedThrottle<0) AND (lMeasuredThrottle<0)))) THEN
		lThrottleArbitrationDelta := ABS(RequestedThrottle) - ABS(lMeasuredThrottle);
		IF (lThrottleArbitrationDelta>lThrottleArbitrationAllowableDelta) THEN
			lProposedThrottle := lMeasuredThrottle;
		END_IF
	END_IF
END_IF

                
END_METHOD

METHOD throttleToVelocity : REAL
  VAR_INPUT
    throttle : t_percentage;
  END_VAR
                  // convert from percentage to rpm
throttleToVelocity := throttle*lMaximumVelocity;
                
END_METHOD

METHOD velocityToThrottle : REAL
  VAR_INPUT
    velocity : REAL;
  END_VAR
                  // convert from rpm to percentage
velocityToThrottle := MAX(-1.0,MIN(velocity/lMaximumVelocity,1.0));

                
END_METHOD

METHOD initializeMotor
  VAR_INPUT
    velocity : REFERENCE TO INT;
    status : REFERENCE TO UINT;
    current : REFERENCE TO USINT;
    alarm : REFERENCE TO UINT;
    motorTemperature : REFERENCE TO USINT;
    controllerTemperature : REFERENCE TO SINT;
    batteryCurrent : REFERENCE TO USINT;
    batteryVoltage : REFERENCE TO UINT;
  END_VAR
                  lVelocity.InputReference REF= velocity;
lTPDO1Stuffing.InputReference ref= status;
lCurrent.InputReference ref= current;
lAlarm.InputReference ref= alarm;
lMotorTemperature.InputReference ref= motorTemperature;
lControllerTemperature.InputReference ref= controllerTemperature;
lBatteryCurrent.InputReference ref= batteryCurrent;
lBatteryVoltage.InputReference ref= batteryVoltage;

// lTorque.InputReference

                
END_METHOD

PROPERTY Alarm : UINT
GET
                    Alarm := lAlarm.Value;
                  
END_GET
END_PROPERTY

PROPERTY BatteryCurrent : REAL
GET
                    BatteryCurrent := lBatteryCurrent.Value;

                  
END_GET
END_PROPERTY

PROPERTY BatteryVoltage : REAL
GET
                    BatteryVoltage := lBatteryVoltage.Value;

                  
END_GET
END_PROPERTY

PROPERTY ClearAlarm : BOOL
GET
                    ClearAlarm := lClearAlarm.Value;

                  
END_GET
SET
                    lClearAlarm.Value := ClearAlarm;
                  
END_SET
END_PROPERTY

PROPERTY Control : WORD
GET
                    Control := lControl;
                  
END_GET
END_PROPERTY

PROPERTY ControllerTemperature : REAL
GET
                    ControllerTemperature := lControllerTemperature.Value;

                  
END_GET
END_PROPERTY

(* {attribute 'monitoring' := 'call'} *)
PROPERTY Current : REAL
GET
                    Current := lCurrent.Value;

                  
END_GET
END_PROPERTY

PROPERTY Diagnostic : t_motor_diagnostic
GET
                    Diagnostic := lDiagnostic;
                  
END_GET
SET
                    _Diagnostic := Diagnostic;
                  
END_SET
END_PROPERTY

PROPERTY Enable : BOOL
GET
                    Enable := lEnable.Value;

                  
END_GET
SET
                    lEnable.Value := Enable;
                  
END_SET
END_PROPERTY

PROPERTY EnableFreeWheel : BOOL
GET
                    EnableFreeWheel := lEnableFreeWheel;
                  
END_GET
SET
                    lEnableFreeWheel := EnableFreeWheel;
                  
END_SET
END_PROPERTY

PROPERTY Forward : BOOL
GET
                    Forward := lForward.Value;

                  
END_GET
END_PROPERTY

PROPERTY FreeWheel : BOOL
GET
                    FreeWheel := lFreeWheel;
                  
END_GET
END_PROPERTY

PROPERTY HoldStationary : BOOL
GET
                    HoldStationary := lHoldStationary;
                  
END_GET
SET
                    lHoldStationary := HoldStationary;
                  
END_SET
END_PROPERTY

PROPERTY MaximumVelocity : REAL
GET
                    MaximumVelocity := lMaximumVelocity;

                  
END_GET
END_PROPERTY

PROPERTY MotorTemperature : REAL
GET
                    MotorTemperature := lMotorTemperature.Value;

                  
END_GET
END_PROPERTY

PROPERTY MotorTemperatureEnabled : BOOL
GET
                    IF ((lEnableDiscriminatoryMotorTemperatureControl) AND
	(NOT(lMotorTemperatureEnabledVerified))) THEN
	checkMotorTemperatureEnabled();
END_IF

MotorTemperatureEnabled := lMotorTemperatureEnabled;
                  
END_GET
SET
                    IF (NOT(lEnableDiscriminatoryMotorTemperatureControl)) THEN
	lMotorTemperatureEnabled := MotorTemperatureEnabled;
	RETURN;
END_IF

IF (lMotorTemperatureEnabled<>MotorTemperatureEnabled) THEN
	lMotorTemperatureEnableCANSequence.MotorTemperatureEnabledRequest := MotorTemperatureEnabled;
	lMotorTemperatureEnableCANSequence.start();
//	IF (MotorTemperatureEnabled) THEN
//		requestSDOWrite(TRUE,16#20F1,16#2,cMotorTemperatureType,4);
//	ELSE
//		requestSDOWrite(TRUE,16#20F1,16#2,0,4);
//	END_IF
END_IF

                  
END_SET
END_PROPERTY

PROPERTY NodeState : t_node_state
SET
                    IF (lEnableNMTDetectionTPDO) THEN

	IF (lTPDO1StuffingPrevious<>lTPDO1Stuffing.Value) THEN
		lNMTDetectionTimer.reset();
	END_IF
	lTPDO1StuffingPrevious := lTPDO1Stuffing.Value;
	
	lNMTDetectionTimer.operator();
	IF (NOT(lNMTDetectionTimer.Expired)) THEN
		lNodeState := t_node_state.OPERATIONAL;
		RETURN;
	ELSE
		IF (gSystemPrimary.SystemState.State>=lStartSystemStateScope) THEN
			start();
		END_IF
	END_IF
END_IF

lNodeState := NodeState;

                  
END_SET
END_PROPERTY

PROPERTY RequestedThrottle : t_percentage
GET
                    RequestedThrottle := lRequestedThrottle.Value;

                  
END_GET
SET
                    lRequestedThrottle.Value := RequestedThrottle;
lRequestedThrottle.operator();
                  
END_SET
END_PROPERTY

PROPERTY Reverse : BOOL
GET
                    Reverse := lReverse.Value;

                  
END_GET
END_PROPERTY

PROPERTY Stalled : BOOL
GET
                    Stalled := lStalled;
                  
END_GET
SET
                    IF ((NOT(Stalled)) AND
	(lStallState=cStallStateClearing)) THEN
	lStallState := cStallStateNone;
END_IF
                  
END_SET
END_PROPERTY

PROPERTY StallInput : BOOL
GET
                    StallInput := StallInput;
                  
END_GET
END_PROPERTY

PROPERTY StallState : t_stall_state
GET
                    StallState := lStallState;
                  
END_GET
END_PROPERTY

PROPERTY Stationary : BOOL
GET
                    Stationary := lStationary;
                  
END_GET
END_PROPERTY

PROPERTY TargetSpeed : REAL
GET
                    // returns as RPM not as Hz
TargetSpeed := lTargetSpeed.Value;

                  
END_GET
END_PROPERTY

PROPERTY ThrottleFreeWheelThreshold : t_percentage
GET
                    ThrottleFreeWheelThreshold := lThrottleFreeWheelThreshold;

                  
END_GET
SET
                    lThrottleFreeWheelThreshold := ThrottleFreeWheelThreshold;

                  
END_SET
END_PROPERTY

PROPERTY ThrottleThreshold : t_percentage
GET
                    ThrottleThreshold := lThrottleThreshold;

                  
END_GET
SET
                    lThrottleThreshold := ThrottleThreshold;
                  
END_SET
END_PROPERTY

PROPERTY Torque : REAL
GET
                    Torque := lTorque.Value;
                  
END_GET
END_PROPERTY

PROPERTY TypeToken : t_medium_string
GET
                    TypeToken := 'cMotor';
                  
END_GET
END_PROPERTY

(* {attribute 'monitoring' := 'call'} *)
PROPERTY Velocity : REAL
GET
                    Velocity := lVelocity.Value;

                  
END_GET
END_PROPERTY

PROPERTY VelocityDelta : REAL
GET
                    VelocityDelta := Velocity - throttleToVelocity(TargetSpeed);
                  
END_GET
END_PROPERTY
END_FUNCTION_BLOCK

FUNCTION_BLOCK ControllerMotor150A EXTENDS ControllerMotor
  VAR CONSTANT
    cNominalCurrent : REAL := 150.0;
    cPolePairs : REAL := 2.0;
    cControllerTemperatureInitialCutbackThreshold : REAL := 75.0;
    cControllerTemperatureCutoutThreshold : REAL := 80.0;
    cControllerTemperatureMinimumThreshold : t_percentage := 0.2;
    cMotorTemperatureInitialCutbackThreshold : REAL := 110.0;
    cMotorTemperatureCutoutThreshold : REAL := 120.0;
    cMotorTemperatureMinimumThreshold : t_percentage := 0.2;
    cMotorTemperatureInvalidRange : REAL := 200;
  END_VAR

            ;
          

METHOD initialize
                  lNominalCurrent := cNominalCurrent;
lPolePairs := cPolePairs;

lMotorTemperatureInvalidRange := cMotorTemperatureInvalidRange;
lMotorTemperatureSensorRecovery := cMotorTemperatureInvalidRange;
	
SUPER^.initialize();

lAlarmControllerTemperatureCutback.InitialCutbackThreshold := cControllerTemperatureInitialCutbackThreshold;
lAlarmControllerTemperatureCutback.CutoutThreshold := cControllerTemperatureCutoutThreshold;
lAlarmControllerTemperatureCutback.MinimiumThreshold := cControllerTemperatureMinimumThreshold;

lAlarmMotorTemperatureCutback.InitialCutbackThreshold := cMotorTemperatureInitialCutbackThreshold;
lAlarmMotorTemperatureCutback.CutoutThreshold := cMotorTemperatureCutoutThreshold;
lAlarmMotorTemperatureCutback.MinimiumThreshold := cMotorTemperatureMinimumThreshold;


                
END_METHOD
END_FUNCTION_BLOCK

FUNCTION_BLOCK ControllerMotor400A EXTENDS ControllerMotor
  VAR CONSTANT
    cNominalCurrent : REAL := 400.0;
    cPolePairs : REAL := 3.0;
    cControllerTemperatureInitialCutbackThreshold : REAL := 75.0;
    cControllerTemperatureCutoutThreshold : REAL := 100.0;
    cControllerTemperatureMinimumThreshold : t_percentage := 0.2;
    cMotorTemperatureInitialCutbackThreshold : REAL := 110.0;
    cMotorTemperatureCutoutThreshold : REAL := 160.0;
    cMotorTemperatureMinimumThreshold : t_percentage := 0.2;
    cMotorTemperatureInvalidRange : REAL := 200;
  END_VAR

            ;
          

METHOD initialize
                  lNominalCurrent := cNominalCurrent;
lPolePairs := cPolePairs;

lMotorTemperatureInvalidRange := cMotorTemperatureInvalidRange;
lMotorTemperatureSensorRecovery := cMotorTemperatureInvalidRange;

SUPER^.initialize();

lAlarmControllerTemperatureCutback.InitialCutbackThreshold := cControllerTemperatureInitialCutbackThreshold;
lAlarmControllerTemperatureCutback.CutoutThreshold := cControllerTemperatureCutoutThreshold;
lAlarmControllerTemperatureCutback.MinimiumThreshold := cControllerTemperatureMinimumThreshold;

lAlarmMotorTemperatureCutback.InitialCutbackThreshold := cMotorTemperatureInitialCutbackThreshold;
lAlarmMotorTemperatureCutback.CutoutThreshold := cMotorTemperatureCutoutThreshold;
lAlarmMotorTemperatureCutback.MinimiumThreshold := cMotorTemperatureMinimumThreshold;
                
END_METHOD
END_FUNCTION_BLOCK

FUNCTION_BLOCK ControllerRotaryEncoder EXTENDS CANOpenSlave
  VAR CONSTANT
    cCalibrationValue : UDINT := 16#40000;
    cStepsPerRevolution : UDINT := 16#4000;
  END_VAR
  VAR
    lAngle : ValueObjectRealOffsetScaledInputReferenceUDINT;
    lAngularVelocity : ValueObjectRealScaledOffsetInputReferenceINT;
    lStepsPerRevolution : UDINT := cStepsPerRevolution;
    lSign : REAL := 1.0;
  END_VAR

            ;
          

METHOD initialize
                  lAngle.initializeValueObjectOp(OpSelf,'Angle','Measured angle','radians',cValueStyleConfigurable);
lAngularVelocity.initializeValueObjectOp(OpSelf,'AngVelocity','Measured angular velocity','rad/s',cValueStyleConfigurable);

SUPER^.initialize();

// radians
lAngle.Offset := 0.0 - UDINT_TO_REAL(cCalibrationValue);
lAngle.Scaling := 2.0 * cPi / UDINT_TO_REAL(lStepsPerRevolution) * lSign;

// hz
lAngularVelocity.Offset := 0.0;
lAngularVelocity.Scaling := 1000.0 / UDINT_TO_REAL(lStepsPerRevolution) * lSign;
                
END_METHOD

METHOD operator
                  SUPER^.operator();

                
END_METHOD

METHOD zero
                  requestSDOWrite(TRUE,16#6003,16#0,UDINT_TO_DWORD(cCalibrationValue),4);


	
                
END_METHOD

METHOD initializeRotaryEncoder
  VAR_INPUT
    angle : REFERENCE TO UDINT;
    velocity : REFERENCE TO INT;
  END_VAR
                  lAngle.InputReference REF= angle;
lAngularVelocity.InputReference REF= velocity;


                
END_METHOD

METHOD execute
  VAR_INPUT
    executeContext : POINTER TO ExecuteContext;
  END_VAR
                  IF (executeContext^.matchCommand(sCommandZero)) THEN	
	zero();
	RETURN;
END_IF

SUPER^.execute(executeContext);


                
END_METHOD

METHOD describe
  VAR_INPUT
    executeContext : POINTER TO ExecuteContext;
  END_VAR
                  SUPER^.describe(executeContext);

IF (executeContext^.matchOption(cExecuteOptionSyntax)) THEN
	executeContext^.describeSyntaxExecutable(sCommandZero);
	RETURN;
END_IF



                
END_METHOD

(* {attribute 'monitoring' := 'call'} *)
PROPERTY Angle : REAL
GET
                    Angle := lAngle.Value;
                  
END_GET
END_PROPERTY

PROPERTY AngleObject : REFERENCE TO ValueObjectReal
GET
                    AngleObject ref= lAngle;
                  
END_GET
END_PROPERTY

(* {attribute 'monitoring' := 'call'} *)
PROPERTY AngularVelocity : REAL
GET
                    AngularVelocity := lAngularVelocity.Value;
                  
END_GET
END_PROPERTY

PROPERTY AngularVelocityObject : REFERENCE TO ValueObjectReal
GET
                    AngularVelocityObject ref= lAngularVelocity;
                  
END_GET
END_PROPERTY

PROPERTY Sign : REAL
GET
                    Sign := lSign;
                  
END_GET
SET
                    lSign := Sign;
                  
END_SET
END_PROPERTY

PROPERTY TypeToken : t_medium_string
GET
                    TypeToken := 'cRotary';
                  
END_GET
END_PROPERTY
END_FUNCTION_BLOCK

{attribute 'enable_dynamic_creation'}
FUNCTION_BLOCK ControllerRotaryEncoderRange EXTENDS ControllerRotaryEncoder
  VAR_INPUT
    lTypeSteer : BOOL := FALSE;
  END_VAR
  VAR
    lVRUpper : ValueReferencePersistentReal;
    lUpper : t_persistent_real;
    lRangeError : ReportableAlarm;
    lPosition : ValueObjectPercentage;
    lLowerErrorBound : t_percentage := -1.01;
    lUpperErrorBound : t_percentage := 1.01;
    lFactor : REAL := 2.0;
    lOffset : REAL := -1.0;
  END_VAR

            ;
          

METHOD initialize
                  IF (lTypeSteer) THEN
	lUpper.Identifier := t_persistent_id.cPersistentID_SteerUpper;
	lFactor := 1.0;
	lOffset := 0.0;

	LowerErrorBound := -1.04;
	UpperErrorBound := 1.04;
END_IF

lVRUpper.initializeValueReference(lUpper,NopSelf,'Upper','Angle at upper end of range','radians',cValueStyleParameter);
lUpper.initialize();

lRangeError.initializeState(NopSelf,'',cACSensorRangeError);

lPosition.initializeValueObject(NopSelf,'Position','Position in established range','',cValueStyleConfigurable);

SUPER^.initialize();

IF (lTypeSteer) THEN
	lAlarmCANOpenSlaveModulation.registerServer(gSystemPrimary.Travel.Interlock);

	Upper := 94.0 / 180.0 * cPi;
END_IF

                
END_METHOD

METHOD operator
                  SUPER^.operator();

IF (NOT(lEnabled)) THEN
	lPosition.Value := 0.0;	
	lPosition.operator();
	RETURN;
END_IF

IF (Upper<>0) THEN
	lPosition.Value := (Angle/Upper*lFactor) + lOffset;
ELSE
	lPosition.Value := 0.0;	
END_IF
lPosition.operator();

IF ((lPosition.Value>lUpperErrorBound) OR
	(lPosition.Value<lLowerErrorBound)) THEN
	lRangeError.trigger(FALSE);
END_IF

                
END_METHOD

METHOD setUpper
                  Upper := Angle;
                
END_METHOD

METHOD execute
  VAR_INPUT
    executeContext : POINTER TO ExecuteContext;
  END_VAR
                  IF (executeContext^.matchCommand(sCommandUpper)) THEN	
	setUpper();
	RETURN;
END_IF

SUPER^.execute(executeContext);


                
END_METHOD

METHOD describe
  VAR_INPUT
    executeContext : POINTER TO ExecuteContext;
  END_VAR
                  SUPER^.describe(executeContext);

IF (executeContext^.matchOption(cExecuteOptionSyntax)) THEN
	executeContext^.describeSyntaxExecutable(sCommandUpper);
	RETURN;
END_IF

                
END_METHOD

PROPERTY LowerErrorBound : t_percentage
GET
                    LowerErrorBound := lLowerErrorBound;
                  
END_GET
SET
                    lLowerErrorBound := LowerErrorBound;
                  
END_SET
END_PROPERTY

(* {attribute 'monitoring' := 'call'} *)
PROPERTY Position : t_percentage
GET
                    Position := lPosition.Value;
                  
END_GET
END_PROPERTY

PROPERTY PositionObject : REFERENCE TO ValueObjectPercentage
GET
                    PositionObject ref= lPosition;
                  
END_GET
END_PROPERTY

PROPERTY TypeToken : t_medium_string
GET
                    TypeToken := 'cRotaryRange';
                  
END_GET
END_PROPERTY

PROPERTY Upper : REAL
GET
                    Upper := lUpper.Value;
                  
END_GET
SET
                    lUpper.Value := Upper;
                  
END_SET
END_PROPERTY

PROPERTY UpperErrorBound : t_percentage
GET
                    UpperErrorBound := lUpperErrorBound;
                  
END_GET
SET
                    lUpperErrorBound := UpperErrorBound;
                  
END_SET
END_PROPERTY

PROPERTY UpperObject : REFERENCE TO t_persistent_real
GET
                    UpperObject ref= lUpper;
                  
END_GET
END_PROPERTY
END_FUNCTION_BLOCK

(* FUNCTION_BLOCK ControllerSteer EXTENDS ControllerMotor150A *)
FUNCTION_BLOCK ControllerSteer EXTENDS ControllerMotor

            ;
          

METHOD initialize
                  lTypeSteer := FALSE;

SUPER^.initialize();

lAlarmCANOpenSlaveModulation.registerServer(gSystemPrimary.Travel.Interlock);
lAlarmCANOpenSlaveBlock.registerServer(gSystemPrimary.Travel.Interlock);

lAlarmControllerTemperatureCutback.registerServer(gSystemPrimary.Travel.ChargeInterlock);
lAlarmMotorTemperatureCutback.registerServer(gSystemPrimary.Travel.ChargeInterlock);

lMaximumVelocity := cSteerMotorMaximumVelocityAsHz;

lAlwaysEnable := FALSE;
lAutomaticEnable := TRUE;

                
END_METHOD
END_FUNCTION_BLOCK

FUNCTION_BLOCK ControllerSteerAngle EXTENDS ControllerRotaryEncoderRange

            ;
          

METHOD initialize
                  lUpper.Identifier := t_persistent_id.cPersistentID_SteerUpper;
lFactor := 1.0;
lOffset := 0.0;

LowerErrorBound := -1.04;
UpperErrorBound := 1.04;

SUPER^.initialize();

lAlarmCANOpenSlaveModulation.registerServer(gSystemPrimary.Travel.Interlock);

Upper := 94.0 / 180.0 * cPi;

                
END_METHOD
END_FUNCTION_BLOCK

(* FUNCTION_BLOCK ControllerTrans EXTENDS ControllerMotor400A *)
FUNCTION_BLOCK ControllerTrans EXTENDS ControllerMotor

            ;
          

METHOD initialize
                  lTypeSteer := FALSE;

SUPER^.initialize();

lAlarmCANOpenSlaveModulation.registerServer(gSystemPrimary.Travel.Interlock);
lAlarmCANOpenSlaveBlock.registerServer(gSystemPrimary.Travel.Interlock);

lAlarmControllerTemperatureCutback.registerServer(gSystemPrimary.Travel.ChargeInterlock);
lAlarmMotorTemperatureCutback.registerServer(gSystemPrimary.Travel.ChargeInterlock);

lMaximumVelocity := cTransMotorMaximumVelocityAsHz;

lAlwaysEnable := FALSE;
lAutomaticEnable := TRUE;
lEnableInitializeHold := FALSE;
//lEnableHoldStationary := TRUE;
lInitializeMotorHoldTimer.Period := cInitializeMotorHoldPeriod;

                
END_METHOD
END_FUNCTION_BLOCK

FUNCTION_BLOCK ControllerUInterface EXTENDS CANOpenSlave
  VAR
    lPackProvider : PackProvider;
  END_VAR

            ;
          

METHOD initialize
                  registerOperational(ADR(lPackProvider));

SUPER^.initialize();
SubSystem := cSubsystemUInterface;

lAlarmCANOpenSlaveModulation.registerServer(gSystemPrimary.Travel.Interlock); // foobar - conditional on cabin not radio?
lAlarmCANOpenSlaveModulation.registerServer(gSystemPrimary.Lift.Interlock); // foobar
// lAlarmCANOpenSlaveNotOperational.Override := TRUE; //foobar
// lOverideConnected := TRUE; //foobar

lAlarmCANOpenSlaveNotOperational.InitialSeverity := cSeverityNone;
lAlarmCANOpenSlaveNotOperational.SeverityWarningTimeout := T#250MS;
lAlarmCANOpenSlaveNotOperational.SeverityErrorTimeout := T#1S;
lAlarmCANOpenSlaveNotOperational.SeverityCriticalTimeout := T#5S;

lAlarmCANOpenSlaveAllowableUp.AllowableSystemState := cSystemStateCharging;
lAlarmCANOpenSlaveAllowableUp.UpperSystemStateScope := cSystemStateCharging;
lAlarmCANOpenSlaveAllowableUp.LowerSystemStateScope := cSystemStateCharging;

lStartSystemStateScope := t_system_state.cSystemStatePreparing;
lOperationalSystemStateScopeLower := t_system_state.cSystemStatePreOperational;
lModulationSystemStateScope := t_system_state.cSystemStateOperational;

lModulationSeverity := cSeverityError;


                
END_METHOD

METHOD initializeControllerUInterfacePackProvider
  VAR_INPUT
    packIn1 : REFERENCE TO USINT;
    packIn2 : REFERENCE TO USINT;
    packIn3 : REFERENCE TO USINT;
    packIn4 : REFERENCE TO USINT;
    packIn5 : REFERENCE TO USINT;
    packIn6 : REFERENCE TO USINT;
    packIn7 : REFERENCE TO USINT;
    packIn8 : REFERENCE TO USINT;
    packOut1 : REFERENCE TO USINT;
    packOut2 : REFERENCE TO USINT;
    packOut3 : REFERENCE TO USINT;
    packOut4 : REFERENCE TO USINT;
    packOut5 : REFERENCE TO USINT;
    packOut6 : REFERENCE TO USINT;
    packOut7 : REFERENCE TO USINT;
    packOut8 : REFERENCE TO USINT;
  END_VAR
                  lPackProvider.initializePackProvider(packIn1,
	packIn2,
	packIn3,
	packIn4,
	packIn5,
	packIn6,
	packIn7,
	packIn8,
	packOut1,
	packOut2,
	packOut3,
	packOut4,
	packOut5,
	packOut6,
	packOut7,
	packOut8);

                
END_METHOD

PROPERTY PackProvider : REFERENCE TO PackProvider
GET
                    PackProvider ref= lPackProvider;
                  
END_GET
END_PROPERTY
END_FUNCTION_BLOCK

FUNCTION_BLOCK ControllerUInterfaceCabin EXTENDS ControllerUInterface
  VAR
    lPeripheral : PeripheralPrimary;
    lLift : ValueObjectPercentageInputReferenceSINT;
    lLiftBalanceAB : ValueObjectPercentageInputReferenceSINT;
    lLiftBalanceAD : ValueObjectPercentageInputReferenceSINT;
    lTravel : ValueObjectPercentageInputReferenceSINT;
    lSteer : ValueObjectPercentageInputReferenceSINT;
    lSideshiftAB : ValueObjectPercentageInputReferenceSINT;
    lSideshiftCD : ValueObjectPercentageInputReferenceSINT;
    lTopbeam : ValueObjectPercentageInputReferenceSINT;
    lTwistlockLock : ValueObjectBoolInputReferenceUSINT;
    lTwistlockUnlock : ValueObjectBoolInputReferenceUSINT;
    lSpreaderTelescopingExtend : ValueObjectBoolInputReferenceUSINT;
    lSpreaderTelescopingRetract : ValueObjectBoolInputReferenceUSINT;
    lJoystickInputPresent : ValueObjectBoolInputReferenceUSINT;
    lLiftJoystickInputPresent : ValueObjectBoolInputReferenceUSINT;
    lTravelJoystickInputPresent : ValueObjectBoolInputReferenceUSINT;
    lConfigurationJoystickInputPresent : ValueObjectBoolInputReferenceUSINT;
    lHorn : ValueObjectBoolInputReferenceUSINT;
    lZeroSteerTargetAngle : ValueObjectBoolInputReferenceUSINT;
    lAutomationStart : ValueObjectBoolInputReferenceUSINT;
    lEstopA : ValueObjectBoolInputReferenceUSINT;
    lStopA : ValueObjectBoolInputReferenceUSINT;
    lEmgyA : ValueObjectBoolInputReferenceUSINT;
    lUMFSA : ValueObjectBoolInputReferenceUSINT;
    lEnableBatteryPackA : ValueObjectBoolInputReferenceUSINT;
    lEstopB : ValueObjectBoolInputReferenceUSINT;
    lStopB : ValueObjectBoolInputReferenceUSINT;
    lEmgyB : ValueObjectBoolInputReferenceUSINT;
    lUMFSB : ValueObjectBoolInputReferenceUSINT;
    lEnableBatteryPackB : ValueObjectBoolInputReferenceUSINT;
  END_VAR

            ;
          

METHOD initialize
                  lLift.initializeValueObjectOp(OpSelf,'Lift','Lift control','',cValueStyleConfigurable);
lLiftBalanceAB.initializeValueObjectOp(OpSelf,'LiftBalanceAB','Lift balance AB end control','',cValueStyleConfigurable);
lLiftBalanceAD.initializeValueObjectOp(OpSelf,'LiftBalanceCD','Lift balance CD end control','',cValueStyleConfigurable);
lTravel.initializeValueObjectOp(OpSelf,'Travel','Travel control','',cValueStyleConfigurable);
lSteer.initializeValueObjectOp(OpSelf,'Steer','Steer control','',cValueStyleConfigurable);	
lSideshiftAB.initializeValueObjectOp(OpSelf,'SideshiftAB','Sideshift AB end control','',cValueStyleConfigurable);
lSideshiftCD.initializeValueObjectOp(OpSelf,'SideshiftCD','Sideshift CD end control','',cValueStyleConfigurable);
lTopbeam.initializeValueObjectOp(OpSelf,'Topbeam','Topbeam control','',cValueStyleConfigurable);

lTwistlockLock.initializeValueObjectOp(OpSelf,'TwstLock','TwstLock control','',cValueStyleConfigurable);
lTwistlockLock.Index := 0;

lTwistlockUnlock.initializeValueObjectOp(OpSelf,'TwstUnlock','TwstUnlock control','',cValueStyleConfigurable);
lTwistlockUnlock.Index := 1;

lSpreaderTelescopingExtend.initializeValueObjectOp(OpSelf,'TelscpExtend','Spreader telescoping extend control','',cValueStyleConfigurable);
lSpreaderTelescopingExtend.Index := 2;

lSpreaderTelescopingRetract.initializeValueObjectOp(OpSelf,'TelscpRetract','Spreader telescoping retract control','',cValueStyleConfigurable);
lSpreaderTelescopingRetract.Index := 3;

lJoystickInputPresent.initializeValueObjectOp(OpSelf,'JoyInpPresent','Joystick control input present','',cValueStyleConfigurable);
lJoystickInputPresent.Index := 0;

lLiftJoystickInputPresent.initializeValueObjectOp(OpSelf,'LiftInpPresent','Lift control input present','',cValueStyleConfigurable);
lLiftJoystickInputPresent.Index := 1;

lTravelJoystickInputPresent.initializeValueObjectOp(OpSelf,'TravelInpPresent','Travel control input present','',cValueStyleConfigurable);
lTravelJoystickInputPresent.Index := 2;

lConfigurationJoystickInputPresent.initializeValueObjectOp(OpSelf,'CnfgInpPresent','Configuration control input present','',cValueStyleConfigurable);
lConfigurationJoystickInputPresent.Index := 3;

lHorn.initializeValueObjectOp(OpSelf,'HornReq','Horn control','',cValueStyleConfigurable);
lHorn.Index := 1;

lZeroSteerTargetAngle.initializeValueObjectOp(OpSelf,'ZeroSteerReq','Zero steer control','',cValueStyleConfigurable);
lZeroSteerTargetAngle.Index := 2;

lAutomationStart.initializeValueObjectOp(OpSelf,'AutoStartReq','Automation start control','',cValueStyleConfigurable);
lAutomationStart.Index := 3;

lEstopA.initializeValueObjectOp(OpSelf,'EstopA','Estop A status','',cValueStyleConfigurable);
lEstopA.Index := 0;

lStopA.initializeValueObjectOp(OpSelf,'StopA','Stop A status','',cValueStyleConfigurable);
lStopA.Index := 1;

lEmgyA.initializeValueObjectOp(OpSelf,'EmcyA','Emcy A status','',cValueStyleConfigurable);
lEmgyA.Index := 2;

lUMFSA.initializeValueObjectOp(OpSelf,'UMFSA','UMFS A status','',cValueStyleConfigurable);
lUMFSA.Index := 3;

lEnableBatteryPackA.initializeValueObjectOp(OpSelf,'EnblBatteryPackA','Enable battery pack A control','',cValueStyleConfigurable);
lEnableBatteryPackA.Index := 4;

lEstopB.initializeValueObjectOp(OpSelf,'EstopB','Estop B status','',cValueStyleConfigurable);
lEstopB.Index := 0;

lStopB.initializeValueObjectOp(OpSelf,'StopB','Stop B status','',cValueStyleConfigurable);
lStopB.Index := 1;

lEmgyB.initializeValueObjectOp(OpSelf,'EmcyB','Emcy B status','',cValueStyleConfigurable);
lEmgyB.Index := 2;

lUMFSB.initializeValueObjectOp(OpSelf,'UMFSB','UMFS B status','',cValueStyleConfigurable);
lUMFSB.Index := 3;

lEnableBatteryPackB.initializeValueObjectOp(OpSelf,'EnblBatteryPackB','Enable battery pack B control','',cValueStyleConfigurable);
lEnableBatteryPackB.Index := 4;

SUPER^.initialize();

lPeripheral.initialize();

lHeartbeatTimer.Period := T#1000MS; // foobar

                
END_METHOD

METHOD operator
                  SUPER^.operator();

lPeripheral.operator();

// foobar null values if no valid transmissions

IF (NOT(Connected)) THEN
	lEstopA.Value := FALSE;
	lEstopB.Value := FALSE;
	lStopA.Value := FALSE;
	lStopB.Value := FALSE;
	lEmgyA.Value := FALSE;
	lEmgyB.Value := FALSE;
	lUMFSA.Value := FALSE;
	lUMFSB.Value := FALSE;
	
	lEnableBatteryPackA.Value := TRUE; // foobar
	lEnableBatteryPackB.Value := TRUE; // foobar
	
	RETURN;
END_IF


                
END_METHOD

METHOD initializeControllerUInterfaceCabin
  VAR_INPUT
    packIn1 : REFERENCE TO USINT;
    packIn2 : REFERENCE TO USINT;
    packIn3 : REFERENCE TO USINT;
    packIn4 : REFERENCE TO USINT;
    packIn5 : REFERENCE TO USINT;
    packIn6 : REFERENCE TO USINT;
    packIn7 : REFERENCE TO USINT;
    packIn8 : REFERENCE TO USINT;
    packOut1 : REFERENCE TO USINT;
    packOut2 : REFERENCE TO USINT;
    packOut3 : REFERENCE TO USINT;
    packOut4 : REFERENCE TO USINT;
    packOut5 : REFERENCE TO USINT;
    packOut6 : REFERENCE TO USINT;
    packOut7 : REFERENCE TO USINT;
    packOut8 : REFERENCE TO USINT;
    lift : REFERENCE TO SINT;
    liftBalanceAB : REFERENCE TO SINT;
    liftBalanceAD : REFERENCE TO SINT;
    travel : REFERENCE TO SINT;
    steer : REFERENCE TO SINT;
    sideShiftAB : REFERENCE TO SINT;
    sideShiftCD : REFERENCE TO SINT;
    topbeam : REFERENCE TO SINT;
    spreaderControls : REFERENCE TO USINT;
    controlsPresent : REFERENCE TO USINT;
    binaryControls : REFERENCE TO USINT;
    binaryStateA : REFERENCE TO USINT;
    binaryStateB : REFERENCE TO USINT;
  END_VAR
                  initializeControllerUInterfacePackProvider(
	packIn1,
	packIn2,
	packIn3,
	packIn4,
	packIn5,
	packIn6,
	packIn7,
	packIn8,

	packOut1,
	packOut2,
	packOut3,
	packOut4,
	packOut5,
	packOut6,
	packOut7,
	packOut8);

lLift.InputReference REF= lift;
lLiftBalanceAB.InputReference REF= liftBalanceAB;
lLiftBalanceAD.InputReference REF= liftBalanceAD;
lTravel.InputReference REF= travel;
lSteer.InputReference REF= steer;
lSideshiftAB.InputReference REF= sideShiftAB;
lSideshiftCD.InputReference REF= sideShiftCD;
lTopbeam.InputReference REF= topbeam;

lTwistlockLock.InputReference REF= spreaderControls;
lTwistlockUnlock.InputReference REF= spreaderControls;
lSpreaderTelescopingExtend.InputReference REF= spreaderControls;
lSpreaderTelescopingRetract.InputReference REF= spreaderControls;

lJoystickInputPresent.InputReference REF= controlsPresent;
lLiftJoystickInputPresent.InputReference REF= controlsPresent;
lTravelJoystickInputPresent.InputReference REF= controlsPresent;
lConfigurationJoystickInputPresent.InputReference REF= controlsPresent;
	
lHorn.InputReference REF= binaryControls;
lZeroSteerTargetAngle.InputReference REF= binaryControls;
lAutomationStart.InputReference REF= binaryControls;
	
lEstopA.InputReference REF= binaryStateA;
lEstopB.InputReference REF= binaryStateB;

lStopA.InputReference REF= binaryStateA;
lStopB.InputReference REF= binaryStateB;

lEmgyA.InputReference REF= binaryStateA;
lEmgyB.InputReference REF= binaryStateB;

lUMFSA.InputReference REF= binaryStateA;
lUMFSB.InputReference REF= binaryStateB;

lEnableBatteryPackA.InputReference REF= binaryStateA;
lEnableBatteryPackB.InputReference REF= binaryStateB;

                
END_METHOD

PROPERTY AutomationStart : BOOL
GET
                    AutomationStart := lAutomationStart.Value;


                  
END_GET
END_PROPERTY

PROPERTY Emgy : BOOL
GET
                    Emgy := ((lEmgyA.Value) AND (lEmgyB.Value));

                  
END_GET
END_PROPERTY

PROPERTY Estop : BOOL
GET
                    Estop := ((lEstopA.Value) AND (lEstopB.Value));
	
                  
END_GET
END_PROPERTY

PROPERTY Horn : BOOL
GET
                    Horn := lHorn.Value; 
                  
END_GET
END_PROPERTY

(* {attribute 'monitoring' := 'call'} *)
PROPERTY JoystickInputPresent : BOOL
GET
                    JoystickInputPresent := lJoystickInputPresent.Value;

                  
END_GET
END_PROPERTY

PROPERTY Lift : t_percentage
GET
                    Lift := lLift.Value;

                  
END_GET
END_PROPERTY

PROPERTY LiftBalanceAB : t_percentage
GET
                    LiftBalanceAB := lLiftBalanceAB.Value;

                  
END_GET
END_PROPERTY

PROPERTY LiftBalanceAD : t_percentage
GET
                    LiftBalanceAD := lLiftBalanceAD.Value;

                  
END_GET
END_PROPERTY

(* {attribute 'monitoring' := 'call'} *)
PROPERTY LiftJoystickInputPresent : BOOL
GET
                    LiftJoystickInputPresent := lLiftJoystickInputPresent.Value;

                  
END_GET
END_PROPERTY

PROPERTY SideshiftAB : t_percentage
GET
                    SideshiftAB := lSideshiftAB.Value;

                  
END_GET
END_PROPERTY

PROPERTY SideshiftCD : t_percentage
GET
                    SideshiftCD := lSideshiftCD.Value;

                  
END_GET
END_PROPERTY

PROPERTY SpreaderTelescopingExtend : BOOL
GET
                    SpreaderTelescopingExtend := lSpreaderTelescopingExtend.Value;

                  
END_GET
END_PROPERTY

PROPERTY SpreaderTelescopingRetract : BOOL
GET
                    SpreaderTelescopingRetract := lSpreaderTelescopingRetract.Value;

                  
END_GET
END_PROPERTY

PROPERTY Steer : t_percentage
GET
                    Steer := lSteer.Value;

                  
END_GET
END_PROPERTY

PROPERTY Stop : BOOL
GET
                    Stop := ((lStopA.Value) and (lStopB.Value));

                  
END_GET
END_PROPERTY

PROPERTY Topbeam : t_percentage
GET
                    Topbeam := lTopbeam.Value;

                  
END_GET
END_PROPERTY

(* {attribute 'monitoring' := 'call'} *)
PROPERTY Travel : t_percentage
GET
                    Travel := lTravel.Value;

                  
END_GET
END_PROPERTY

(* {attribute 'monitoring' := 'call'} *)
PROPERTY TravelJoystickInputPresent : BOOL
GET
                    TravelJoystickInputPresent := lTravelJoystickInputPresent.Value;

                  
END_GET
END_PROPERTY

PROPERTY TwistlockLock : BOOL
GET
                    TwistlockLock := lTwistlockLock.Value;

                  
END_GET
END_PROPERTY

PROPERTY TwistlockUnlock : BOOL
GET
                    TwistlockUnlock := lTwistlockUnlock.Value;

                  
END_GET
END_PROPERTY

PROPERTY TypeToken : t_medium_string
GET
                    TypeToken := 'cDisplay';
                  
END_GET
END_PROPERTY

PROPERTY UMFS : BOOL
GET
                    UMFS := ((lUMFSA.Value) AND (lUMFSB.Value));

                  
END_GET
END_PROPERTY

PROPERTY ZeroSteerTargetAngle : BOOL
GET
                    ZeroSteerTargetAngle := lZeroSteerTargetAngle.Value;

                  
END_GET
END_PROPERTY

PROPERTY EnableBatteryPack : BOOL
GET
                    EnableBatteryPack := ((lEnableBatteryPackA.Value) AND (lEnableBatteryPackB.Value));

                  
END_GET
END_PROPERTY

PROPERTY Peripheral : REFERENCE TO Peripheral
GET
                    Peripheral ref= lPeripheral;
                  
END_GET
END_PROPERTY
END_FUNCTION_BLOCK

FUNCTION_BLOCK ControllerUInterfaceRadio EXTENDS ControllerUInterface
  VAR CONSTANT
    cBatteryTimerPeriod : t_ms_time := TIME#1m0s0ms;
    cRadioBatteryBit : USINT := 1;  (* gRadioXState *)
    cRadioTimedStopBit : USINT := 2;  (* gRadioXState *)
    cRadioEmgyBit : USINT := 3;  (* gRadioXState *)
    cRadioSafetyCANOpenBit : USINT := 6;  (* gRadioXState *)
    cRadioStopBit : USINT := 7;  (* gRadioXState *)
    cRadioStartBit : USINT := 0;  (* gRadioXSwitch1 *)
    cRadioTwistlockUnlockBit : USINT := 1;  (* gRadioXSwitch1 *)
    cRadioTwistlockLockBit : USINT := 2;  (* gRadioXSwitch1 *)
    cRadioHornBit : USINT := 7;  (* gRadioXSwitch1 *)
    cRadioButtonBit : USINT := 0;  (* gRadioXSwitch2 *)
    cRadioTiltBit : USINT := 4;  (* gRadioXPackIn1 *)
    cStartPeriod : t_ms_time := TIME#1s0ms;
  END_VAR
  VAR
    _DummyPackIn : USINT := 0;
    lLeftXaxis : ValueObjectPercentageInputReferenceUSINTJoystick;
    lLeftYaxis : ValueObjectPercentageInputReferenceUSINTJoystick;
    lRightXaxis : ValueObjectPercentageInputReferenceUSINTJoystick;
    lRightYaxis : ValueObjectPercentageInputReferenceUSINTJoystick;
    lRightRotation : ValueObjectPercentageInputReferenceUSINTJoystick;
    lBattery : ValueObjectBoolInputReferenceUSINT;
    lButton : ValueObjectBoolInputReferenceUSINT;
    lStop : ValueObjectBoolInputReferenceUSINT;
    lSafetyCANOpen : ValueObjectBoolInputReferenceUSINT;
    lTImedStop : ValueObjectBoolInputReferenceUSINT;
    lEmgy : ValueObjectBoolInputReferenceUSINT;
    lTilt : ValueObjectBoolInputReferenceUSINT;
    lStartButton : ValueObjectBoolInputReferenceUSINT;
    lHorn : ValueObjectBoolInputReferenceUSINT;
    lTwistlockLock : ValueObjectBoolInputReferenceUSINT;
    lTwistlockUnlock : ValueObjectBoolInputReferenceUSINT;
    lBatteryTimer : t_timer;
  END_VAR

            ;
          

METHOD emergencyHandler
  VAR_INPUT
    info : t_canopen_emcy;
  END_VAR
  VAR
    eid : t_radio_emcy_id;
    first : BOOL;
  END_VAR
                  first := emergencyRegisterAdd(info);

eid := WORD_TO_INT(info.EMCY_ERROR_CODE);

CASE eid OF
	cEMCY_none,
	cEMCY_RECOVERED_FROM_BUS_OFF:
		RETURN;

	cEMCY_PDO_LENGTH_EXCEEDED,
	cEMCY_GENERIC_ERROR,
	cEMCY_CURRENT,
	cEMCY_CURRENT_DEVICE_INPUT_SIDE,
	cEMCY_CURRENT_INSIDE_THE_DEVICE,
	cEMCY_CURRENT_DEVICE_OUTPUT_SIDE,
	cEMCY_CURRENT_AT_OUTPUTS_TOO_HIGH,
	cEMCY_SHORT_CIRCUIT_AT_OUTPUTS,
	cEMCY_LOAD_DUMP_AT_OUTPUTS,
	cEMCY_VOLTAGE,
	cEMCY_MAINS_VOLTAGE,
	cEMCY_INPUT_VOLTAGE_TOO_HIGH,
	cEMCY_INPUT_VOLTAGE_TOO_LOW,
	cEMCY_VOLTAGE_INSIDE_THE_DEVICE,
	cEMCY_INTERNAL_VOLTAGE_TOO_HIGH,
	cEMCY_INTERNAL_VOLTAGE_TOO_LOW,
	cEMCY_OUTPUT_VOLTAGE,
	cEMCY_OUTPUT_VOLTAGE_TOO_HIGH,
	cEMCY_OUTPUT_VOLTAGE_TOO_LOW,
	cEMCY_TEMPERATURE,
	cEMCY_AMBIENT_TEMPERATURE,
	cEMCY_DEVICE_TEMPERATURE,
	cEMCY_DEVICE_HARDWARE,
	cEMCY_DEVICE_SOFTWARE,
	cEMCY_INTERNAL_SOFTWARE,
	cEMCY_USER_SOFTWARE,
	cEMCY_DATA_SET,
	cEMCY_ADDITIONAL_MODULES,
	cEMCY_MONITORING,
	cEMCY_COMMUNICATION,
	cEMCY_PROTOCOL_ERROR,
	cEMCY_EXTERNAL_ERROR,
	cEMCY_ADDITIONAL_FUNCTIONS,
	cEMCY_DEVICE_SPECIFIC,
	cEMCY_PDO_NOT_PROCESSED_DUE_TO_LENGTH_ERROR,
	cEMCY_TRANSMIT_COB_ID_COLLISION,
	cEMCY_CAN_IN_ERROR_PASSIVE_MODE,	
	cEMCY_CAN_OVERRUN,
	cEMCY_LIFE_GUARD_ERROR_OR_HEARTBEAT_ERROR:
		lAlarmCANOpenSlaveNotify.triggerWithContext(INT_TO_WORD(eid));
		RETURN;
	
//		lAlarmCANOpenSlaveBlock.triggerWithContext(INT_TO_WORD(eid));
	
//		lAlarmCANOpenSlaveStop.triggerWithContext(INT_TO_WORD(eid));
END_CASE

lAlarmCANOpenSlaveNotify.triggerWithContext(INT_TO_WORD(eid));

                
END_METHOD

METHOD initialize
                  lLeftXaxis.initializeValueObjectOp(OpSelf,'LeftX','Left joystick X-axis control','',cValueStyleConfigurable);
lLeftYaxis.initializeValueObjectOp(OpSelf,'LeftY','Left joystick Y-axis control','',cValueStyleConfigurable);
lLeftYaxis.Alpha := 1.0;
lRightXaxis.initializeValueObjectOp(OpSelf,'RightA','Right joystick X-axis control','',cValueStyleConfigurable);
lRightYaxis.initializeValueObjectOp(OpSelf,'RightY','Right joystick Y-axis control','',cValueStyleConfigurable);
lRightRotation.initializeValueObjectOp(OpSelf,'RightRot','Right joystick rotation control','',cValueStyleConfigurable);

lBattery.Index := cRadioBatteryBit;
lBattery.initializeValueObjectOp(OpSelf,'Battery','Radio battery status','',cValueStyleConfigurable);

lButton.Index := cRadioButtonBit;
lButton.initializeValueObjectOp(OpSelf,'Button','Left joystick button control','',cValueStyleConfigurable);

lEmgy.Index := cRadioEmgyBit;
lEmgy.initializeValueObjectOp(OpSelf,'Emcy','Radio emcy status','',cValueStyleConfigurable);

lHorn.Index := cRadioHornBit;
lHorn.initializeValueObjectOp(OpSelf,'HornReq','Radio horn control','',cValueStyleConfigurable);

lSafetyCANOpen.Index := cRadioSafetyCANOpenBit;
lSafetyCANOpen.initializeValueObjectOp(OpSelf,'Safety','Radio safety status','',cValueStyleConfigurable);

lStartButton.Index := cRadioStartBit;
lStartButton.initializeValueObjectOp(OpSelf,'StartButton','Radio start control','',cValueStyleConfigurable);

lStop.Index := cRadioStopBit;
lStop.initializeValueObjectOp(OpSelf,'Stop','Radio stop status','',cValueStyleConfigurable);

lTImedStop.Index := cRadioTimedStopBit;
lTImedStop.initializeValueObjectOp(OpSelf,'TimedStop','Radio timed-stop status','',cValueStyleConfigurable);

lTilt.Index := cRadioTiltBit;
lTilt.initializeValueObjectOp(OpSelf,'Tilt','Radio tilt status','',cValueStyleConfigurable);

lTwistlockLock.Index := cRadioTwistlockLockBit;
lTwistlockLock.initializeValueObjectOp(OpSelf,'TwstLock','Radio twistlock lock control','',cValueStyleConfigurable);

lTwistlockUnlock.Index := cRadioTwistlockUnlockBit;
lTwistlockUnlock.initializeValueObjectOp(OpSelf,'TwstUnlock','Radio twistlock unlock control','',cValueStyleConfigurable);

SUPER^.initialize();

lBatteryTimer.initialize();
lBatteryTimer.Period := cBatteryTimerPeriod;
lBatteryTimer.Enable := TRUE;
                
END_METHOD

METHOD operator
                  SUPER^.operator();

IF (lBattery.Value) THEN
	lBatteryTimer.operator();
	IF (lBatteryTimer.lExpired) THEN
		//gMessageManager.register(lCode:=t_message_code.cMCAdviseUIBattery);
		lBatteryTimer.reset();
	END_IF
ELSE
	lBatteryTimer.reset();
END_IF

IF (lTilt.Value) THEN
	;
END_IF

                
END_METHOD

METHOD initializeControllerUInterfaceRadio
  VAR_INPUT
    packIn1 : REFERENCE TO USINT;
    packIn2 : REFERENCE TO USINT;
    packIn3 : REFERENCE TO USINT;
    packIn4 : REFERENCE TO USINT;
    packOut1 : REFERENCE TO USINT;
    packOut2 : REFERENCE TO USINT;
    packOut3 : REFERENCE TO USINT;
    packOut4 : REFERENCE TO USINT;
    packOut5 : REFERENCE TO USINT;
    packOut6 : REFERENCE TO USINT;
    packOut7 : REFERENCE TO USINT;
    packOut8 : REFERENCE TO USINT;
    leftXaxis : REFERENCE TO USINT;
    leftYaxis : REFERENCE TO USINT;
    rightXaxis : REFERENCE TO USINT;
    rightYaxis : REFERENCE TO USINT;
    rightRotation : REFERENCE TO USINT;
    state : REFERENCE TO USINT;
    switch1 : REFERENCE TO USINT;
    switch2 : REFERENCE TO USINT;
  END_VAR
                  initializeControllerUInterfacePackProvider(
	packIn1,
	packIn2,
	packIn3,
	packIn4,
	_DummyPackIn,
	_DummyPackIn,
	_DummyPackIn,
	_DummyPackIn,

	packOut1,
	packOut2,
	packOut3,
	packOut4,
	packOut5,
	packOut6,
	packOut7,
	packOut8);

lLeftXaxis.InputReference REF= leftXaxis;
lLeftYaxis.InputReference REF= leftYaxis;
lRightXaxis.InputReference REF= rightXaxis;
lRightYaxis.InputReference REF= rightYaxis;
lRightRotation.InputReference REF= rightRotation;

lBattery.InputReference REF= state;
lTImedStop.InputReference REF= state;
lEmgy.InputReference REF= state;
lSafetyCANOpen.InputReference REF= state;
lStop.InputReference REF= state;

lStartButton.InputReference REF= switch1;
lTwistlockLock.InputReference REF= switch1;
lTwistlockUnlock.InputReference REF= switch1;	
lHorn.InputReference REF= switch1;
lButton.InputReference REF= switch2;
lTilt.InputReference REF= switch1;

                
END_METHOD

PROPERTY AutomationStart : BOOL
GET
                    AutomationStart := FALSE;

IF (gSystemPrimary.ProgrammedMovementControl.Enabled) THEN
	AutomationStart := Button;
END_IF


                  
END_GET
END_PROPERTY

PROPERTY Battery : BOOL
GET
                    Battery := lBattery.Value;

                  
END_GET
END_PROPERTY

PROPERTY Button : BOOL
GET
                    Button := lButton.Value;
                  
END_GET
END_PROPERTY

PROPERTY Emgy : BOOL
GET
                    Emgy := lEmgy.Value;
                  
END_GET
END_PROPERTY

PROPERTY Horn : BOOL
GET
                    Horn := lHorn.Value;
                  
END_GET
END_PROPERTY

(* {attribute 'monitoring' := 'call'} *)
PROPERTY JoystickInputPresent : BOOL
GET
                    JoystickInputPresent := ((lLeftXaxis.InputPresent) OR
	(lLeftYaxis.InputPresent) OR
	(lRightXaxis.InputPresent) OR
	(lRightYaxis.InputPresent) OR
	(lRightRotation.InputPresent));

                  
END_GET
END_PROPERTY

(* {attribute 'monitoring' := 'call'} *)
PROPERTY LeftJoystickInputPresent : BOOL
GET
                    LeftJoystickInputPresent := ((lLeftXaxis.InputPresent) OR
	(lLeftYaxis.InputPresent));

                  
END_GET
END_PROPERTY

PROPERTY LeftXaxis : t_percentage
GET
                    LeftXaxis := lLeftXaxis.Value;
                  
END_GET
END_PROPERTY

(* {attribute 'monitoring' := 'call'} *)
PROPERTY LeftYaxis : t_percentage
GET
                    LeftYaxis := lLeftYaxis.Value;
                  
END_GET
END_PROPERTY

PROPERTY SafetyCANOpen : BOOL
GET
                    SafetyCANOpen := lSafetyCANOpen.Value;
                  
END_GET
END_PROPERTY

(* {attribute 'monitoring' := 'call'} *)
PROPERTY RightJoystickInputPresent : BOOL
GET
                    RightJoystickInputPresent := ((lRightXaxis.InputPresent) OR
	(lRightYaxis.InputPresent) OR
	(lRightRotation.InputPresent));

                  
END_GET
END_PROPERTY

PROPERTY RightRotation : t_percentage
GET
                    RightRotation := lRightRotation.Value;
                  
END_GET
END_PROPERTY

PROPERTY RightXaxis : t_percentage
GET
                    RightXaxis := lRightXaxis.Value;
                  
END_GET
END_PROPERTY

PROPERTY RightYaxis : t_percentage
GET
                    RightYaxis := lRightYaxis.Value;
                  
END_GET
END_PROPERTY

PROPERTY StartButton : BOOL
GET
                    StartButton := lStartButton.Value;
                  
END_GET
END_PROPERTY

PROPERTY Stop : BOOL
GET
                    Stop := lStop.Value;
                  
END_GET
END_PROPERTY

PROPERTY StopObject : REFERENCE TO ValueObjectBool
GET
                    StopObject REF= lStop;

                  
END_GET
END_PROPERTY

PROPERTY TimedStop : BOOL
GET
                    TimedStop := lTimedStop.Value;
                  
END_GET
END_PROPERTY

PROPERTY TwistlockLock : BOOL
GET
                    TwistlockLock := lTwistlockLock.Value;
                  
END_GET
END_PROPERTY

PROPERTY TwistlockUnlock : BOOL
GET
                    TwistlockUnlock := lTwistlockUnlock.Value;
                  
END_GET
END_PROPERTY

PROPERTY TypeToken : t_medium_string
GET
                    TypeToken := 'cRadio';
                  
END_GET
END_PROPERTY

PROPERTY ZeroSteerTargetAngle : BOOL
GET
                    ZeroSteerTargetAngle := FALSE;

IF (NOT(gSystemPrimary.ProgrammedMovementControl.Enabled)) THEN
	ZeroSteerTargetAngle := Button;
END_IF


                  
END_GET
END_PROPERTY

PROPERTY EnableBatteryPack : BOOL
GET
                    EnableBatteryPack := TRUE;

                  
END_GET
END_PROPERTY
END_FUNCTION_BLOCK

FUNCTION_BLOCK CheckMotorTemperatureEnableCANMessage EXTENDS SDOReadCANMessage
  VAR
    lMotorTemperatureEnabled : BOOL;
  END_VAR

            
          

METHOD initialize
                  SUPER^.initialize();

lSDORead.INDEX := 16#20F1;
lSDORead.SUBINDEX := 1;

lSDODReadDataLength := 4;

                
END_METHOD

METHOD sdoReadHandler
                  lMotorTemperatureEnabled := (lSDOReadData<>0);

                
END_METHOD

PROPERTY MotorTemperatureEnabled : BOOL
GET
                    MotorTemperatureEnabled := lMotorTemperatureEnabled;
                  
END_GET
END_PROPERTY
END_FUNCTION_BLOCK

FUNCTION_BLOCK DisableWriteMotorControllerCANMessage EXTENDS SDOWriteCANMessage

            
          

METHOD initialize
                  SUPER^.initialize();

lSDOWrite.INDEX := 16#1010;
lSDOWrite.SUBINDEX := 1;

lSDOWriteData := 16#534F4C43;

                
END_METHOD
END_FUNCTION_BLOCK

FUNCTION_BLOCK EditMotorTemperatureEnableCANMessage EXTENDS SDOWriteCANMessage
  VAR
    lMotorTemperatureEnabled : BOOL := TRUE;
  END_VAR

            
          

METHOD initialize
                  SUPER^.initialize();

lSDOWrite.INDEX := 16#20F1;
lSDOWrite.SUBINDEX := 1;
lSDOWrite.DATALENGTH := 4;

IF (lMotorTemperatureEnabled) THEN
	lSDOWriteData := 4;
ELSE
	lSDOWriteData := 0;	
END_IF

                
END_METHOD

METHOD start
                  IF (lMotorTemperatureEnabled) THEN
	lSDOWriteData := 4;
ELSE
	lSDOWriteData := 0;	
END_IF

SUPER^.start();
                
END_METHOD

PROPERTY MotorTemperatureEnabled : BOOL
GET
                    MotorTemperatureEnabled := lMotorTemperatureEnabled;
                  
END_GET
SET
                    lMotorTemperatureEnabled := MotorTemperatureEnabled;
                  
END_SET
END_PROPERTY
END_FUNCTION_BLOCK

FUNCTION_BLOCK EnableWriteMotorControllerCANMessage EXTENDS SDOWriteCANMessage

            
          

METHOD initialize
                  SUPER^.initialize();

lSDOWrite.INDEX := 16#1010;
lSDOWrite.SUBINDEX := 1;
lSDOWrite.DATALENGTH := 4;

lSDOWriteData := 16#4E45504F;

                
END_METHOD
END_FUNCTION_BLOCK

FUNCTION_BLOCK MotorTemperatureEnableCANSequence EXTENDS CANMessageSequence
  VAR
    lPreCheck : CheckMotorTemperatureEnableCANMessage;
    lEnableWrite : EnableWriteMotorControllerCANMessage;
    lEdit : EditMotorTemperatureEnableCANMessage;
    lDisableWrite : DisableWriteMotorControllerCANMessage;
    lPostCheck : CheckMotorTemperatureEnableCANMessage;
    lMotorTemperatureEnabledPreCheck : BOOL;
    lMotorTemperatureEnabledRequest : BOOL;
    lMotorTemperatureEnabledPostCheck : BOOL;
  END_VAR

            
          

METHOD initialize
                  registerMessage(ADR(lPreCheck));
registerMessage(ADR(lEnableWrite));
registerMessage(ADR(lEdit));
registerMessage(ADR(lDisableWrite));
registerMessage(ADR(lPostCheck));

SUPER^.initialize();
                
END_METHOD

METHOD operator
  VAR
    b : BOOL;
  END_VAR
                  IF ((NOT(Enabled)) OR (Running)) THEN
	RETURN;
END_IF

SUPER^.operator();

IF (lPreCheck.Finished) THEN
	lMotorTemperatureEnabledPreCheck := lPreCheck.MotorTemperatureEnabled;
END_IF

IF (lPostCheck.Finished) THEN
	lMotorTemperatureEnabledPostCheck := lPostCheck.MotorTemperatureEnabled;
END_IF

                
END_METHOD

METHOD start
                  lEdit.MotorTemperatureEnabled := lMotorTemperatureEnabledRequest;

SUPER^.start();

                
END_METHOD

PROPERTY MotorTemperatureEnabledPostCheck : BOOL
GET
                    MotorTemperatureEnabledPostCheck := lMotorTemperatureEnabledPostCheck;
                  
END_GET
END_PROPERTY

PROPERTY MotorTemperatureEnabledPreCheck : BOOL
GET
                    MotorTemperatureEnabledPreCheck := lMotorTemperatureEnabledPreCheck;
                  
END_GET
END_PROPERTY

PROPERTY MotorTemperatureEnabledRequest : BOOL
GET
                    MotorTemperatureEnabledRequest := lMotorTemperatureEnabledRequest;
                  
END_GET
SET
                    lMotorTemperatureEnabledRequest := MotorTemperatureEnabledRequest;
                  
END_SET
END_PROPERTY
END_FUNCTION_BLOCK

FUNCTION_BLOCK FunctionalMode
  VAR
    lEnabled : BOOL := FALSE;  (* lMaintainer: StandardMaintainer; *)
    lAvailable : BOOL := FALSE;
    lMode : t_functional_mode := cFunctionalModeAny;
    lState : t_mode_state := cModeStateInactive;
  END_VAR

            ;
          

METHOD enter : BOOL
                  lState := cModeStateActive;
enter := TRUE;

                
END_METHOD

METHOD initialize
                  

                
END_METHOD

METHOD leave : BOOL
                  lState := cModeStateInactive;
leave := TRUE;
                
END_METHOD

PROPERTY Active : BOOL
GET
                    Active := (lState=cModeStateActive);
                  
END_GET
END_PROPERTY

PROPERTY Available : BOOL
GET
                    Available := lAvailable;
                  
END_GET
SET
                    lAvailable := Available;
                  
END_SET
END_PROPERTY

PROPERTY Enabled : BOOL
GET
                    Enabled := ((lEnabled) and (lAvailable));
                  
END_GET
SET
                    lEnabled := Enabled;
                  
END_SET
END_PROPERTY

PROPERTY Mode : t_functional_mode
GET
                    Mode := lMode;
                  
END_GET
END_PROPERTY

PROPERTY State : t_mode_state
GET
                    State := lState;
                  
END_GET
END_PROPERTY
END_FUNCTION_BLOCK

FUNCTION_BLOCK FunctionalModeControl EXTENDS NonOperationalParticleSet
  VAR
    lFunctionalModeDefault : FunctionalModeDefault;
    lFunctionalModeTravel : FunctionalModeTravel;
    lFunctionalModeLift : FunctionalModeLift;
    lMode : REFERENCE TO FunctionalMode;
    lDiagnostic : t_functional_diagnostic;
    lRequested : BOOL := FALSE;
  END_VAR

            ;
          

METHOD enableAndRequest : t_functional_diagnostic
  VAR_INPUT
    requested : t_functional_mode;
  END_VAR
  VAR
    previous : BOOL;
    mode : REFERENCE TO FunctionalMode;
  END_VAR
                  IF (requested=cFunctionalModeAny) THEN
	enableAndRequest := cFunctionalDiagnosticOK;
	RETURN;
END_IF

mode REF= getMode(requested);
previous := mode.Enabled;

mode.Enabled := TRUE;
enableAndRequest := request(requested);
IF (enableAndRequest>cFunctionalDiagnosticNotYetActive) THEN
	mode.Enabled := previous;
END_IF
                
END_METHOD

METHOD getMode : REFERENCE TO FunctionalMode
  VAR_INPUT
    mode : t_functional_mode;
  END_VAR
                  getMode REF= lFunctionalModeDefault;
	
CASE mode OF		
	cFunctionalModeDefault:
		getMode REF= lFunctionalModeDefault;	
	cFunctionalModeTravel:
		getMode REF= lFunctionalModeTravel;
	cFunctionalModeLift:
		getMode REF= lFunctionalModeLift;
END_CASE

                
END_METHOD

METHOD initialize
                  SUPER^.initialize();

lFunctionalModeDefault.Available := TRUE;
lFunctionalModeDefault.Enabled := TRUE;
lFunctionalModeDefault.initialize();

lFunctionalModeTravel.Available := TRUE;
lFunctionalModeTravel.Enabled := TRUE;
lFunctionalModeTravel.initialize();

lFunctionalModeLift.Available := TRUE;
lFunctionalModeLift.Enabled := TRUE;
lFunctionalModeLift.initialize();

lMode REF= lFunctionalModeDefault;
                
END_METHOD

METHOD leave : t_functional_diagnostic
                  leave := request(cFunctionalModeDefault);

                
END_METHOD

METHOD operator
                  lRequested := FALSE;
lDiagnostic := cFunctionalDiagnosticOK;

enableAndRequest(gSystemPrimary.UInterface.FunctionalModeRequest);

IF (lMode.State=cModeStateEntering) THEN
	IF (NOT(lMode.enter())) THEN
		lDiagnostic := cFunctionalDiagnosticNotYetActive;
		RETURN;
	END_IF
	
	RETURN;
END_IF

IF (lMode.State=cModeStateExiting) THEN
	IF (NOT(lMode.leave())) THEN
		lDiagnostic := cFunctionalDiagnosticWaitingToExit;
		RETURN;
	END_IF
	
	RETURN;
END_IF

                
END_METHOD

METHOD request : t_functional_diagnostic
  VAR_INPUT
    requested : t_functional_mode;
  END_VAR
  VAR
    mode : REFERENCE TO FunctionalMode;
  END_VAR
                  IF (requested=cFunctionalModeAny) THEN
	lDiagnostic := cFunctionalDiagnosticOK;
	request := lDiagnostic;
	RETURN;
END_IF

IF (CurrentMode=requested) THEN
	IF (NOT(lMode.enter())) THEN
		//gMessageManager.register(lCode:=cMCAdviseFunctionalModeNotYetActive);
		lDiagnostic := cFunctionalDiagnosticNotYetActive;
		request := lDiagnostic;
		RETURN;		
	END_IF
	
	lDiagnostic := cFunctionalDiagnosticOK;
	request := lDiagnostic;
	RETURN;
END_IF

IF (lRequested) THEN
	//gMessageManager.register(lCode:=cMCAdviseFunctionalModeRace);
	lDiagnostic := cFunctionalDiagnosticRace;
	request := lDiagnostic;
	RETURN;	
END_IF

mode REF= getMode(requested);

IF (NOT(mode.Enabled)) THEN
	//gMessageManager.register(lCode:=cMCAdviseFunctionalModeIllegalRequest);
	lDiagnostic := cFunctionalDiagnosticNotEnabled;
	request := lDiagnostic;
	RETURN;
END_IF

